LIN {X 0,Y 134.923,Z 410.508,A -85,B 0,C 180,E1 -24681.385,E2 -24681.385} C_VEL
LIN {X 0,Y 135.857,Z 404.738,A -85,B 0,C 180,E1 -24688.426,E2 -24688.426} C_VEL
LIN {X 0,Y 136.109,Z 403.534,A -85,B 0,C 180,E1 -24689.947,E2 -24689.947} C_VEL
LIN {X 0,Y 136.386,Z 403.497,A -85,B 0,C 180,E1 -24691.018,E2 -24691.018} C_VEL
LIN {X 0,Y 136.277,Z 403.499,A -85,B 0,C 180,E1 -24694.562,E2 -24694.562} C_VEL
LIN {X 0,Y 136.081,Z 403.534,A -85,B 0,C 180,E1 -24699.223,E2 -24699.223} C_VEL
LIN {X 0,Y 136.001,Z 403.539,A -85,B 0,C 180,E1 -24703.658,E2 -24703.658} C_VEL
LIN {X 0,Y 136.007,Z 403.542,A -85,B 0,C 180,E1 -24707.797,E2 -24707.797} C_VEL
LIN {X 0,Y 136.029,Z 403.534,A -85,B 0,C 180,E1 -24711.684,E2 -24711.684} C_VEL
LIN {X 0,Y 136.087,Z 403.533,A -85,B 0,C 180,E1 -24715.721,E2 -24715.721} C_VEL
LIN {X 0,Y 136.149,Z 403.524,A -85,B 0,C 180,E1 -24722.317,E2 -24722.317} C_VEL
LIN {X 0,Y 136.247,Z 403.508,A -85,B 0,C 180,E1 -24728.833,E2 -24728.833} C_VEL
LIN {X 0,Y 136.275,Z 403.507,A -85,B 0,C 180,E1 -24735.057,E2 -24735.057} C_VEL
LIN {X 0,Y 136.447,Z 403.483,A -85,B 0,C 180,E1 -24738.138,E2 -24738.138} C_VEL
LIN {X 0,Y 136.555,Z 403.474,A -85,B 0,C 180,E1 -24741.118,E2 -24741.118} C_VEL
LIN {X 0,Y 137.136,Z 403.404,A -85,B 0,C 180,E1 -24750,E2 -24750} C_VEL
LIN {X 0,Y 136.595,Z 403.469,A -85,B 0,C 180,E1 -24758.879,E2 -24758.879} C_VEL
LIN {X 0,Y 136.493,Z 403.477,A -85,B 0,C 180,E1 -24761.954,E2 -24761.954} C_VEL
LIN {X 0,Y 136.276,Z 403.509,A -85,B 0,C 180,E1 -24768.025,E2 -24768.025} C_VEL
LIN {X 0,Y 136.229,Z 403.51,A -85,B 0,C 180,E1 -24771.779,E2 -24771.779} C_VEL
LIN {X 0,Y 136.103,Z 403.528,A -85,B 0,C 180,E1 -24778.616,E2 -24778.616} C_VEL
LIN {X 0,Y 136.081,Z 403.533,A -85,B 0,C 180,E1 -24784.618,E2 -24784.618} C_VEL
LIN {X 0,Y 136.052,Z 403.532,A -85,B 0,C 180,E1 -24789.208,E2 -24789.208} C_VEL
LIN {X 0,Y 135.999,Z 403.544,A -85,B 0,C 180,E1 -24793.657,E2 -24793.657} C_VEL
LIN {X 0,Y 135.985,Z 403.541,A -85,B 0,C 180,E1 -24797.788,E2 -24797.788} C_VEL
LIN {X 0,Y 136.029,Z 403.54,A -85,B 0,C 180,E1 -24801.684,E2 -24801.684} C_VEL
LIN {X 0,Y 136.058,Z 403.53,A -85,B 0,C 180,E1 -24805.738,E2 -24805.738} C_VEL
LIN {X 0,Y 136.149,Z 403.524,A -85,B 0,C 180,E1 -24812.317,E2 -24812.317} C_VEL
LIN {X 0,Y 136.246,Z 403.515,A -85,B 0,C 180,E1 -24818.833,E2 -24818.833} C_VEL
LIN {X 0,Y 136.291,Z 403.507,A -85,B 0,C 180,E1 -24825.058,E2 -24825.058} C_VEL
LIN {X 0,Y 136.503,Z 403.481,A -85,B 0,C 180,E1 -24828.115,E2 -24828.115} C_VEL
LIN {X 0,Y 136.61,Z 403.461,A -85,B 0,C 180,E1 -24831.121,E2 -24831.121} C_VEL
LIN {X 0,Y 137.136,Z 403.396,A -85,B 0,C 180,E1 -24840,E2 -24840} C_VEL
LIN {X 0,Y 136.61,Z 403.463,A -85,B 0,C 180,E1 -24848.878,E2 -24848.878} C_VEL
LIN {X 0,Y 136.494,Z 403.482,A -85,B 0,C 180,E1 -24851.958,E2 -24851.958} C_VEL
LIN {X 0,Y 136.253,Z 403.507,A -85,B 0,C 180,E1 -24858.028,E2 -24858.028} C_VEL
LIN {X 0,Y 136.199,Z 403.52,A -85,B 0,C 180,E1 -24861.749,E2 -24861.749} C_VEL
LIN {X 0,Y 136.101,Z 403.531,A -85,B 0,C 180,E1 -24868.616,E2 -24868.616} C_VEL
LIN {X 0,Y 136.079,Z 403.529,A -85,B 0,C 180,E1 -24874.618,E2 -24874.618} C_VEL
LIN {X 0,Y 136.063,Z 403.536,A -85,B 0,C 180,E1 -24879.214,E2 -24879.214} C_VEL
LIN {X 0,Y 136.313,Z 403.581,A -85,B 0,C 180,E1 -24885.161,E2 -24885.161} C_VEL
LIN {X 0,Y 137.773,Z 409.554,A -85,B 0,C 180,E1 -24891.226,E2 -24891.226} C_VEL
LIN {X 0,Y 139.191,Z 414.655,A -85,B 0,C 180,E1 -24896.261,E2 -24896.261} C_VEL
LIN {X 0,Y 139.438,Z 416.517,A -85,B 0,C 180,E1 -24898.049,E2 -24898.049} C_VEL
LIN {X 0,Y 136.371,Z 425.684,A -85,B 0,C 180,E1 -24907.203,E2 -24907.203} C_VEL
LIN {X 0,Y 136.444,Z 432.258,A -85,B 0,C 180,E1 -24913.927,E2 -24913.927} C_VEL
LIN {X 0,Y 136.598,Z 432.809,A -85,B 0,C 180,E1 -24914.234,E2 -24914.234} C_VEL
LIN {X 0,Y 137.103,Z 444.83,A -85,B 0,C 180,E1 -24915.94,E2 -24915.94} C_VEL
LIN {X 0,Y 138.431,Z 457.423,A -85,B 0,C 180,E1 -24918.283,E2 -24918.283} C_VEL
LIN {X 0,Y 139.405,Z 464.257,A -85,B 0,C 180,E1 -24919.837,E2 -24919.837} C_VEL
LIN {X 0,Y 139.365,Z 473.819,A -85,B 0,C 180,E1 -24922.758,E2 -24922.758} C_VEL
LIN {X 0,Y 139.631,Z 483.352,A -85,B 0,C 180,E1 -24926.393,E2 -24926.393} C_VEL
LIN {X 0,Y 140.17,Z 490.988,A -85,B 0,C 180,E1 -24930,E2 -24930} C_VEL
LIN {X 0,Y 140.133,Z 494.562,A -85,B 0,C 180,E1 -24932.156,E2 -24932.156} C_VEL
LIN {X 0,Y 139.561,Z 497.394,A -85,B 0,C 180,E1 -24934.332,E2 -24934.332} C_VEL
LIN {X 0,Y 138.249,Z 501.754,A -85,B 0,C 180,E1 -24938.773,E2 -24938.773} C_VEL
LIN {X 0,Y 137.884,Z 506.27,A -85,B 0,C 180,E1 -24944.765,E2 -24944.765} C_VEL
LIN {X 0,Y 139.405,Z 509.537,A -85,B 0,C 180,E1 -24950.665,E2 -24950.665} C_VEL
LIN {X 0,Y 142.833,Z 511.707,A -85,B 0,C 180,E1 -24956.286,E2 -24956.286} C_VEL
LIN {X 0,Y 148.061,Z 512.881,A -85,B 0,C 180,E1 -24961.476,E2 -24961.476} C_VEL
LIN {X 0,Y 154.895,Z 513.043,A -85,B 0,C 180,E1 -24966.146,E2 -24966.146} C_VEL
LIN {X 0,Y 163.095,Z 512.189,A -85,B 0,C 180,E1 -24970.269,E2 -24970.269} C_VEL
LIN {X 0,Y 172.559,Z 510.242,A -85,B 0,C 180,E1 -24973.819,E2 -24973.819} C_VEL
LIN {X 0,Y 177.592,Z 508.832,A -85,B 0,C 180,E1 -24975.425,E2 -24975.425} C_VEL
LIN {X 0,Y 179.65,Z 508.061,A -85,B 0,C 180,E1 -24976.364,E2 -24976.364} C_VEL
LIN {X 0,Y 180.102,Z 507.363,A -85,B 0,C 180,E1 -24977.853,E2 -24977.853} C_VEL
LIN {X 0,Y 178.396,Z 506.566,A -85,B 0,C 180,E1 -24980.926,E2 -24980.926} C_VEL
LIN {X 0,Y 176.25,Z 506.125,A -85,B 0,C 180,E1 -24983.264,E2 -24983.264} C_VEL
LIN {X 0,Y 172.11,Z 506.046,A -85,B 0,C 180,E1 -24985.132,E2 -24985.132} C_VEL
LIN {X 0,Y 165.014,Z 505.378,A -85,B 0,C 180,E1 -24987.834,E2 -24987.834} C_VEL
LIN {X 0,Y 158.459,Z 503.885,A -85,B 0,C 180,E1 -24990.799,E2 -24990.799} C_VEL
LIN {X 0,Y 154.466,Z 502.309,A -85,B 0,C 180,E1 -24992.936,E2 -24992.936} C_VEL
LIN {X 0,Y 149.037,Z 499.137,A -85,B 0,C 180,E1 -24996.37,E2 -24996.37} C_VEL
LIN {X 0,Y 148.231,Z 498.488,A -85,B 0,C 180,E1 -24996.975,E2 -24996.975} C_VEL
LIN {X 0,Y 145.275,Z 496.327,A -85,B 0,C 180,E1 -24998.773,E2 -24998.773} C_VEL
LIN {X 0,Y 139.381,Z 491.98,A -85,B 0,C 180,E1 -25001.462,E2 -25001.462} C_VEL
LIN {X 0,Y 134.104,Z 486.835,A -85,B 0,C 180,E1 -25004.254,E2 -25004.254} C_VEL
LIN {X 0,Y 132.202,Z 483.453,A -85,B 0,C 180,E1 -25006.182,E2 -25006.182} C_VEL
LIN {X 0,Y 130.071,Z 474.061,A -85,B 0,C 180,E1 -25011.455,E2 -25011.455} C_VEL
LIN {X 0,Y 129.418,Z 465.891,A -85,B 0,C 180,E1 -25015.328,E2 -25015.328} C_VEL
LIN {X 0,Y 129.469,Z 454.926,A -85,B 0,C 180,E1 -25019.611,E2 -25019.611} C_VEL
LIN {X 0,Y 129.665,Z 446.445,A -85,B 0,C 180,E1 -25022.33,E2 -25022.33} C_VEL
LIN {X 0,Y 129.871,Z 436.015,A -85,B 0,C 180,E1 -25025.045,E2 -25025.045} C_VEL
LIN {X 0,Y 129.845,Z 430.527,A -85,B 0,C 180,E1 -25026.215,E2 -25026.215} C_VEL
LIN {X 0,Y 128.67,Z 421.434,A -85,B 0,C 180,E1 -25027.782,E2 -25027.782} C_VEL
LIN {X 0,Y 127.321,Z 417.429,A -85,B 0,C 180,E1 -25032.756,E2 -25032.756} C_VEL
LIN {X 0,Y 127.758,Z 411.164,A -85,B 0,C 180,E1 -25040.743,E2 -25040.743} C_VEL
LIN {X 0,Y 128.612,Z 405.807,A -85,B 0,C 180,E1 -25047.602,E2 -25047.602} C_VEL
LIN {X 0,Y 128.89,Z 404.435,A -85,B 0,C 180,E1 -25049.39,E2 -25049.39} C_VEL
LIN {X 0,Y 129.242,Z 404.372,A -85,B 0,C 180,E1 -25052.942,E2 -25052.942} C_VEL
LIN {X 0,Y 129.073,Z 404.406,A -85,B 0,C 180,E1 -25056.795,E2 -25056.795} C_VEL
LIN {X 0,Y 128.985,Z 404.415,A -85,B 0,C 180,E1 -25060.833,E2 -25060.833} C_VEL
LIN {X 0,Y 128.924,Z 404.425,A -85,B 0,C 180,E1 -25065.127,E2 -25065.127} C_VEL
LIN {X 0,Y 128.944,Z 404.42,A -85,B 0,C 180,E1 -25069.735,E2 -25069.735} C_VEL
LIN {X 0,Y 128.983,Z 404.419,A -85,B 0,C 180,E1 -25074.818,E2 -25074.818} C_VEL
LIN {X 0,Y 129.036,Z 404.406,A -85,B 0,C 180,E1 -25080.647,E2 -25080.647} C_VEL
LIN {X 0,Y 129.111,Z 404.398,A -85,B 0,C 180,E1 -25087.602,E2 -25087.602} C_VEL
LIN {X 0,Y 129.16,Z 404.395,A -85,B 0,C 180,E1 -25090.944,E2 -25090.944} C_VEL
LIN {X 0,Y 129.369,Z 404.364,A -85,B 0,C 180,E1 -25097.922,E2 -25097.922} C_VEL
LIN {X 0,Y 129.48,Z 404.356,A -85,B 0,C 180,E1 -25100.628,E2 -25100.628} C_VEL
LIN {X 0,Y 130.091,Z 404.281,A -85,B 0,C 180,E1 -25110,E2 -25110} C_VEL
LIN {X 0,Y 129.52,Z 404.351,A -85,B 0,C 180,E1 -25119.368,E2 -25119.368} C_VEL
LIN {X 0,Y 129.397,Z 404.359,A -85,B 0,C 180,E1 -25122.548,E2 -25122.548} C_VEL
LIN {X 0,Y 129.188,Z 404.391,A -85,B 0,C 180,E1 -25129.051,E2 -25129.051} C_VEL
LIN {X 0,Y 129.138,Z 404.395,A -85,B 0,C 180,E1 -25132.393,E2 -25132.393} C_VEL
LIN {X 0,Y 129.037,Z 404.406,A -85,B 0,C 180,E1 -25139.373,E2 -25139.373} C_VEL
LIN {X 0,Y 128.994,Z 404.418,A -85,B 0,C 180,E1 -25145.189,E2 -25145.189} C_VEL
LIN {X 0,Y 128.952,Z 404.42,A -85,B 0,C 180,E1 -25150.845,E2 -25150.845} C_VEL
LIN {X 0,Y 128.917,Z 404.424,A -85,B 0,C 180,E1 -25155.129,E2 -25155.129} C_VEL
LIN {X 0,Y 128.937,Z 404.423,A -85,B 0,C 180,E1 -25159.738,E2 -25159.738} C_VEL
LIN {X 0,Y 128.962,Z 404.416,A -85,B 0,C 180,E1 -25164.83,E2 -25164.83} C_VEL
LIN {X 0,Y 129.052,Z 404.41,A -85,B 0,C 180,E1 -25170.651,E2 -25170.651} C_VEL
LIN {X 0,Y 129.109,Z 404.402,A -85,B 0,C 180,E1 -25177.727,E2 -25177.727} C_VEL
LIN {X 0,Y 129.165,Z 404.393,A -85,B 0,C 180,E1 -25180.945,E2 -25180.945} C_VEL
LIN {X 0,Y 129.42,Z 404.363,A -85,B 0,C 180,E1 -25187.814,E2 -25187.814} C_VEL
LIN {X 0,Y 129.532,Z 404.344,A -85,B 0,C 180,E1 -25190.632,E2 -25190.632} C_VEL
LIN {X 0,Y 130.092,Z 404.274,A -85,B 0,C 180,E1 -25200,E2 -25200} C_VEL
LIN {X 0,Y 129.532,Z 404.344,A -85,B 0,C 180,E1 -25209.368,E2 -25209.368} C_VEL
LIN {X 0,Y 129.395,Z 404.367,A -85,B 0,C 180,E1 -25212.548,E2 -25212.548} C_VEL
LIN {X 0,Y 129.161,Z 404.393,A -85,B 0,C 180,E1 -25219.055,E2 -25219.055} C_VEL
LIN {X 0,Y 129.109,Z 404.402,A -85,B 0,C 180,E1 -25222.398,E2 -25222.398} C_VEL
LIN {X 0,Y 129.036,Z 404.411,A -85,B 0,C 180,E1 -25229.373,E2 -25229.373} C_VEL
LIN {X 0,Y 128.994,Z 404.411,A -85,B 0,C 180,E1 -25235.19,E2 -25235.19} C_VEL
LIN {X 0,Y 129.011,Z 404.412,A -85,B 0,C 180,E1 -25240.822,E2 -25240.822} C_VEL
LIN {X 0,Y 129.309,Z 404.45,A -85,B 0,C 180,E1 -25245.452,E2 -25245.452} C_VEL
LIN {X 0,Y 130.772,Z 410.28,A -85,B 0,C 180,E1 -25251.707,E2 -25251.707} C_VEL
LIN {X 0,Y 131.968,Z 414.402,A -85,B 0,C 180,E1 -25256.001,E2 -25256.001} C_VEL
LIN {X 0,Y 132.301,Z 416.274,A -85,B 0,C 180,E1 -25257.913,E2 -25257.913} C_VEL
LIN {X 0,Y 129.245,Z 425.368,A -85,B 0,C 180,E1 -25267.627,E2 -25267.627} C_VEL
LIN {X 0,Y 129.433,Z 431.429,A -85,B 0,C 180,E1 -25274.247,E2 -25274.247} C_VEL
LIN {X 0,Y 129.83,Z 432.468,A -85,B 0,C 180,E1 -25275.124,E2 -25275.124} C_VEL
LIN {X 0,Y 130.443,Z 444.677,A -85,B 0,C 180,E1 -25276.986,E2 -25276.986} C_VEL
LIN {X 0,Y 131.772,Z 456.247,A -85,B 0,C 180,E1 -25279.242,E2 -25279.242} C_VEL
LIN {X 0,Y 132.84,Z 463.183,A -85,B 0,C 180,E1 -25280.868,E2 -25280.868} C_VEL
LIN {X 0,Y 132.91,Z 473.806,A -85,B 0,C 180,E1 -25284.31,E2 -25284.31} C_VEL
LIN {X 0,Y 133.271,Z 482.289,A -85,B 0,C 180,E1 -25287.734,E2 -25287.734} C_VEL
LIN {X 0,Y 133.772,Z 488.453,A -85,B 0,C 180,E1 -25290.753,E2 -25290.753} C_VEL
LIN {X 0,Y 133.736,Z 492.301,A -85,B 0,C 180,E1 -25293.165,E2 -25293.165} C_VEL
LIN {X 0,Y 132.794,Z 495.697,A -85,B 0,C 180,E1 -25296.076,E2 -25296.076} C_VEL
LIN {X 0,Y 131.466,Z 501.251,A -85,B 0,C 180,E1 -25302.347,E2 -25302.347} C_VEL
LIN {X 0,Y 132.063,Z 505.446,A -85,B 0,C 180,E1 -25308.621,E2 -25308.621} C_VEL
LIN {X 0,Y 134.734,Z 508.516,A -85,B 0,C 180,E1 -25314.664,E2 -25314.664} C_VEL
LIN {X 0,Y 139.237,Z 510.545,A -85,B 0,C 180,E1 -25320.315,E2 -25320.315} C_VEL
LIN {X 0,Y 145.557,Z 511.616,A -85,B 0,C 180,E1 -25325.409,E2 -25325.409} C_VEL
LIN {X 0,Y 153.433,Z 511.739,A -85,B 0,C 180,E1 -25329.887,E2 -25329.887} C_VEL
LIN {X 0,Y 162.537,Z 510.85,A -85,B 0,C 180,E1 -25333.776,E2 -25333.776} C_VEL
LIN {X 0,Y 172.611,Z 508.879,A -85,B 0,C 180,E1 -25337.129,E2 -25337.129} C_VEL
LIN {X 0,Y 172.25,Z 508.109,A -85,B 0,C 180,E1 -25339.246,E2 -25339.246} C_VEL
LIN {X 0,Y 170.406,Z 507.374,A -85,B 0,C 180,E1 -25341.783,E2 -25341.783} C_VEL
LIN {X 0,Y 166.321,Z 506.966,A -85,B 0,C 180,E1 -25343.731,E2 -25343.731} C_VEL
LIN {X 0,Y 156.711,Z 505.324,A -85,B 0,C 180,E1 -25347.441,E2 -25347.441} C_VEL
LIN {X 0,Y 152.284,Z 503.896,A -85,B 0,C 180,E1 -25349.492,E2 -25349.492} C_VEL
LIN {X 0,Y 144.308,Z 499.738,A -85,B 0,C 180,E1 -25354.004,E2 -25354.004} C_VEL
LIN {X 0,Y 139.337,Z 495.438,A -85,B 0,C 180,E1 -25357.772,E2 -25357.772} C_VEL
LIN {X 0,Y 134.671,Z 489.065,A -85,B 0,C 180,E1 -25362.538,E2 -25362.538} C_VEL
LIN {X 0,Y 132.202,Z 483.453,A -85,B 0,C 180,E1 -25366.182,E2 -25366.182} C_VEL
LIN {X 0,Y 130.599,Z 479.926,A -85,B 0,C 180,E1 -25368.095,E2 -25368.095} C_VEL
LIN {X 0,Y 126.875,Z 473.349,A -85,B 0,C 180,E1 -25370.916,E2 -25370.916} C_VEL
LIN {X 0,Y 123.597,Z 466.089,A -85,B 0,C 180,E1 -25373.694,E2 -25373.694} C_VEL
LIN {X 0,Y 122.777,Z 461.607,A -85,B 0,C 180,E1 -25375.504,E2 -25375.504} C_VEL
LIN {X 0,Y 122.912,Z 450.852,A -85,B 0,C 180,E1 -25379.591,E2 -25379.591} C_VEL
LIN {X 0,Y 122.991,Z 441.44,A -85,B 0,C 180,E1 -25382.457,E2 -25382.457} C_VEL
LIN {X 0,Y 123.165,Z 430.67,A -85,B 0,C 180,E1 -25385.116,E2 -25385.116} C_VEL
LIN {X 0,Y 121.993,Z 421.815,A -85,B 0,C 180,E1 -25386.696,E2 -25386.696} C_VEL
LIN {X 0,Y 120.327,Z 417.894,A -85,B 0,C 180,E1 -25391.796,E2 -25391.796} C_VEL
LIN {X 0,Y 120.699,Z 410.831,A -85,B 0,C 180,E1 -25401.307,E2 -25401.307} C_VEL
LIN {X 0,Y 121.656,Z 405.488,A -85,B 0,C 180,E1 -25408.513,E2 -25408.513} C_VEL
LIN {X 0,Y 121.964,Z 405.294,A -85,B 0,C 180,E1 -25411.24,E2 -25411.24} C_VEL
LIN {X 0,Y 122.046,Z 405.279,A -85,B 0,C 180,E1 -25416.274,E2 -25416.274} C_VEL
LIN {X 0,Y 121.91,Z 405.295,A -85,B 0,C 180,E1 -25421.457,E2 -25421.457} C_VEL
LIN {X 0,Y 121.874,Z 405.303,A -85,B 0,C 180,E1 -25428.561,E2 -25428.561} C_VEL
LIN {X 0,Y 121.935,Z 405.297,A -85,B 0,C 180,E1 -25434.804,E2 -25434.804} C_VEL
LIN {X 0,Y 121.943,Z 405.288,A -85,B 0,C 180,E1 -25439.827,E2 -25439.827} C_VEL
LIN {X 0,Y 121.986,Z 405.288,A -85,B 0,C 180,E1 -25446.215,E2 -25446.215} C_VEL
LIN {X 0,Y 122.05,Z 405.277,A -85,B 0,C 180,E1 -25449.787,E2 -25449.787} C_VEL
LIN {X 0,Y 122.242,Z 405.25,A -85,B 0,C 180,E1 -25456.704,E2 -25456.704} C_VEL
LIN {X 0,Y 122.409,Z 405.236,A -85,B 0,C 180,E1 -25460.081,E2 -25460.081} C_VEL
LIN {X 0,Y 122.602,Z 405.209,A -85,B 0,C 180,E1 -25466.714,E2 -25466.714} C_VEL
LIN {X 0,Y 123.045,Z 405.159,A -85,B 0,C 180,E1 -25470,E2 -25470} C_VEL
LIN {X 0,Y 122.45,Z 405.231,A -85,B 0,C 180,E1 -25476.591,E2 -25476.591} C_VEL
LIN {X 0,Y 122.449,Z 405.231,A -85,B 0,C 180,E1 -25479.915,E2 -25479.915} C_VEL
LIN {X 0,Y 122.289,Z 405.245,A -85,B 0,C 180,E1 -25483.29,E2 -25483.29} C_VEL
LIN {X 0,Y 122.076,Z 405.273,A -85,B 0,C 180,E1 -25490.208,E2 -25490.208} C_VEL
LIN {X 0,Y 121.998,Z 405.287,A -85,B 0,C 180,E1 -25493.781,E2 -25493.781} C_VEL
LIN {X 0,Y 121.943,Z 405.288,A -85,B 0,C 180,E1 -25500.173,E2 -25500.173} C_VEL
LIN {X 0,Y 121.913,Z 405.297,A -85,B 0,C 180,E1 -25506.189,E2 -25506.189} C_VEL
LIN {X 0,Y 121.885,Z 405.302,A -85,B 0,C 180,E1 -25511.444,E2 -25511.444} C_VEL
LIN {X 0,Y 121.866,Z 405.3,A -85,B 0,C 180,E1 -25518.565,E2 -25518.565} C_VEL
LIN {X 0,Y 121.914,Z 405.294,A -85,B 0,C 180,E1 -25524.797,E2 -25524.797} C_VEL
LIN {X 0,Y 121.94,Z 405.295,A -85,B 0,C 180,E1 -25529.828,E2 -25529.828} C_VEL
LIN {X 0,Y 121.985,Z 405.287,A -85,B 0,C 180,E1 -25536.215,E2 -25536.215} C_VEL
LIN {X 0,Y 122.053,Z 405.28,A -85,B 0,C 180,E1 -25539.788,E2 -25539.788} C_VEL
LIN {X 0,Y 122.288,Z 405.253,A -85,B 0,C 180,E1 -25546.709,E2 -25546.709} C_VEL
LIN {X 0,Y 122.458,Z 405.228,A -85,B 0,C 180,E1 -25550.086,E2 -25550.086} C_VEL
LIN {X 0,Y 122.612,Z 405.211,A -85,B 0,C 180,E1 -25556.714,E2 -25556.714} C_VEL
LIN {X 0,Y 123.046,Z 405.151,A -85,B 0,C 180,E1 -25560,E2 -25560} C_VEL
LIN {X 0,Y 122.459,Z 405.228,A -85,B 0,C 180,E1 -25566.591,E2 -25566.591} C_VEL
LIN {X 0,Y 122.458,Z 405.226,A -85,B 0,C 180,E1 -25569.914,E2 -25569.914} C_VEL
LIN {X 0,Y 122.265,Z 405.254,A -85,B 0,C 180,E1 -25573.293,E2 -25573.293} C_VEL
LIN {X 0,Y 122.051,Z 405.282,A -85,B 0,C 180,E1 -25580.212,E2 -25580.212} C_VEL
LIN {X 0,Y 121.984,Z 405.288,A -85,B 0,C 180,E1 -25583.784,E2 -25583.784} C_VEL
LIN {X 0,Y 121.942,Z 405.296,A -85,B 0,C 180,E1 -25590.174,E2 -25590.174} C_VEL
LIN {X 0,Y 121.916,Z 405.296,A -85,B 0,C 180,E1 -25596.192,E2 -25596.192} C_VEL
LIN {X 0,Y 122.073,Z 405.273,A -85,B 0,C 180,E1 -25603.698,E2 -25603.698} C_VEL
LIN {X 0,Y 122.297,Z 405.278,A -85,B 0,C 180,E1 -25605.79,E2 -25605.79} C_VEL
LIN {X 0,Y 123.862,Z 411.27,A -85,B 0,C 180,E1 -25612.596,E2 -25612.596} C_VEL
LIN {X 0,Y 125.082,Z 415.684,A -85,B 0,C 180,E1 -25617.438,E2 -25617.438} C_VEL
LIN {X 0,Y 123.854,Z 419.021,A -85,B 0,C 180,E1 -25621.163,E2 -25621.163} C_VEL
LIN {X 0,Y 122.14,Z 429.42,A -85,B 0,C 180,E1 -25633.28,E2 -25633.28} C_VEL
LIN {X 0,Y 123.086,Z 431.907,A -85,B 0,C 180,E1 -25636.089,E2 -25636.089} C_VEL
LIN {X 0,Y 123.909,Z 445.534,A -85,B 0,C 180,E1 -25638.343,E2 -25638.343} C_VEL
LIN {X 0,Y 125.437,Z 456.947,A -85,B 0,C 180,E1 -25640.731,E2 -25640.731} C_VEL
LIN {X 0,Y 126.306,Z 462.085,A -85,B 0,C 180,E1 -25642.004,E2 -25642.004} C_VEL
LIN {X 0,Y 126.499,Z 472.65,A -85,B 0,C 180,E1 -25645.619,E2 -25645.619} C_VEL
LIN {X 0,Y 127.048,Z 481.337,A -85,B 0,C 180,E1 -25649.368,E2 -25649.368} C_VEL
LIN {X 0,Y 127.589,Z 487.079,A -85,B 0,C 180,E1 -25652.368,E2 -25652.368} C_VEL
LIN {X 0,Y 127.359,Z 489.743,A -85,B 0,C 180,E1 -25654.193,E2 -25654.193} C_VEL
LIN {X 0,Y 126.124,Z 493.904,A -85,B 0,C 180,E1 -25658.008,E2 -25658.008} C_VEL
LIN {X 0,Y 125.217,Z 499.381,A -85,B 0,C 180,E1 -25664.63,E2 -25664.63} C_VEL
LIN {X 0,Y 125.873,Z 502.645,A -85,B 0,C 180,E1 -25669.573,E2 -25669.573} C_VEL
LIN {X 0,Y 128.681,Z 506.08,A -85,B 0,C 180,E1 -25675.908,E2 -25675.908} C_VEL
LIN {X 0,Y 133.412,Z 508.447,A -85,B 0,C 180,E1 -25681.789,E2 -25681.789} C_VEL
LIN {X 0,Y 139.98,Z 509.929,A -85,B 0,C 180,E1 -25687.048,E2 -25687.048} C_VEL
LIN {X 0,Y 148.135,Z 510.49,A -85,B 0,C 180,E1 -25691.622,E2 -25691.622} C_VEL
LIN {X 0,Y 157.516,Z 510.086,A -85,B 0,C 180,E1 -25695.552,E2 -25695.552} C_VEL
LIN {X 0,Y 165.089,Z 509.134,A -85,B 0,C 180,E1 -25698.046,E2 -25698.046} C_VEL
LIN {X 0,Y 164.109,Z 508.288,A -85,B 0,C 180,E1 -25700.431,E2 -25700.431} C_VEL
LIN {X 0,Y 160.623,Z 507.645,A -85,B 0,C 180,E1 -25702.225,E2 -25702.225} C_VEL
LIN {X 0,Y 150.747,Z 505.383,A -85,B 0,C 180,E1 -25705.982,E2 -25705.982} C_VEL
LIN {X 0,Y 144.014,Z 502.65,A -85,B 0,C 180,E1 -25709.176,E2 -25709.176} C_VEL
LIN {X 0,Y 137.971,Z 498.908,A -85,B 0,C 180,E1 -25712.713,E2 -25712.713} C_VEL
LIN {X 0,Y 132.851,Z 494.204,A -85,B 0,C 180,E1 -25716.624,E2 -25716.624} C_VEL
LIN {X 0,Y 128.073,Z 487.269,A -85,B 0,C 180,E1 -25721.607,E2 -25721.607} C_VEL
LIN {X 0,Y 125.145,Z 480.069,A -85,B 0,C 180,E1 -25726.192,E2 -25726.192} C_VEL
LIN {X 0,Y 123.428,Z 471.271,A -85,B 0,C 180,E1 -25730.992,E2 -25730.992} C_VEL
LIN {X 0,Y 122.777,Z 461.607,A -85,B 0,C 180,E1 -25735.504,E2 -25735.504} C_VEL
LIN {X 0,Y 122.092,Z 457.024,A -85,B 0,C 180,E1 -25737.205,E2 -25737.205} C_VEL
LIN {X 0,Y 120.672,Z 452.145,A -85,B 0,C 180,E1 -25738.65,E2 -25738.65} C_VEL
LIN {X 0,Y 117.434,Z 441.865,A -85,B 0,C 180,E1 -25741.172,E2 -25741.172} C_VEL
LIN {X 0,Y 116.552,Z 436.486,A -85,B 0,C 180,E1 -25742.448,E2 -25742.448} C_VEL
LIN {X 0,Y 116.494,Z 434.675,A -85,B 0,C 180,E1 -25742.895,E2 -25742.895} C_VEL
LIN {X 0,Y 116.409,Z 429.421,A -85,B 0,C 180,E1 -25744.112,E2 -25744.112} C_VEL
LIN {X 0,Y 115.383,Z 422.175,A -85,B 0,C 180,E1 -25745.462,E2 -25745.462} C_VEL
LIN {X 0,Y 113.392,Z 418.319,A -85,B 0,C 180,E1 -25750.716,E2 -25750.716} C_VEL
LIN {X 0,Y 113.674,Z 410.429,A -85,B 0,C 180,E1 -25761.968,E2 -25761.968} C_VEL
LIN {X 0,Y 114.475,Z 406.23,A -85,B 0,C 180,E1 -25768.162,E2 -25768.162} C_VEL
LIN {X 0,Y 114.898,Z 406.174,A -85,B 0,C 180,E1 -25771.09,E2 -25771.09} C_VEL
LIN {X 0,Y 114.922,Z 406.17,A -85,B 0,C 180,E1 -25777.343,E2 -25777.343} C_VEL
LIN {X 0,Y 114.811,Z 406.177,A -85,B 0,C 180,E1 -25782.729,E2 -25782.729} C_VEL
LIN {X 0,Y 114.797,Z 406.185,A -85,B 0,C 180,E1 -25787.667,E2 -25787.667} C_VEL
LIN {X 0,Y 114.8,Z 406.18,A -85,B 0,C 180,E1 -25792.737,E2 -25792.737} C_VEL
LIN {X 0,Y 114.869,Z 406.17,A -85,B 0,C 180,E1 -25798.933,E2 -25798.933} C_VEL
LIN {X 0,Y 114.949,Z 406.163,A -85,B 0,C 180,E1 -25806.507,E2 -25806.507} C_VEL
LIN {X 0,Y 115.016,Z 406.158,A -85,B 0,C 180,E1 -25812.21,E2 -25812.21} C_VEL
LIN {X 0,Y 115.254,Z 406.12,A -85,B 0,C 180,E1 -25817.333,E2 -25817.333} C_VEL
LIN {X 0,Y 115.369,Z 406.112,A -85,B 0,C 180,E1 -25823.002,E2 -25823.002} C_VEL
LIN {X 0,Y 115.996,Z 406.037,A -85,B 0,C 180,E1 -25830,E2 -25830} C_VEL
LIN {X 0,Y 115.391,Z 406.11,A -85,B 0,C 180,E1 -25836.996,E2 -25836.996} C_VEL
LIN {X 0,Y 115.308,Z 406.114,A -85,B 0,C 180,E1 -25842.785,E2 -25842.785} C_VEL
LIN {X 0,Y 115.036,Z 406.156,A -85,B 0,C 180,E1 -25847.786,E2 -25847.786} C_VEL
LIN {X 0,Y 114.968,Z 406.161,A -85,B 0,C 180,E1 -25853.514,E2 -25853.514} C_VEL
LIN {X 0,Y 114.87,Z 406.17,A -85,B 0,C 180,E1 -25861.068,E2 -25861.068} C_VEL
LIN {X 0,Y 114.803,Z 406.178,A -85,B 0,C 180,E1 -25867.747,E2 -25867.747} C_VEL
LIN {X 0,Y 114.794,Z 406.185,A -85,B 0,C 180,E1 -25872.72,E2 -25872.72} C_VEL
LIN {X 0,Y 114.789,Z 406.18,A -85,B 0,C 180,E1 -25877.663,E2 -25877.663} C_VEL
LIN {X 0,Y 114.789,Z 406.186,A -85,B 0,C 180,E1 -25882.743,E2 -25882.743} C_VEL
LIN {X 0,Y 114.863,Z 406.177,A -85,B 0,C 180,E1 -25888.937,E2 -25888.937} C_VEL
LIN {X 0,Y 114.948,Z 406.164,A -85,B 0,C 180,E1 -25896.507,E2 -25896.507} C_VEL
LIN {X 0,Y 115.022,Z 406.151,A -85,B 0,C 180,E1 -25902.211,E2 -25902.211} C_VEL
LIN {X 0,Y 115.288,Z 406.124,A -85,B 0,C 180,E1 -25907.257,E2 -25907.257} C_VEL
LIN {X 0,Y 115.395,Z 406.108,A -85,B 0,C 180,E1 -25909.472,E2 -25909.472} C_VEL
LIN {X 0,Y 115.539,Z 406.093,A -85,B 0,C 180,E1 -25916.512,E2 -25916.512} C_VEL
LIN {X 0,Y 115.998,Z 406.029,A -85,B 0,C 180,E1 -25920,E2 -25920} C_VEL
LIN {X 0,Y 115.4,Z 406.106,A -85,B 0,C 180,E1 -25926.996,E2 -25926.996} C_VEL
LIN {X 0,Y 115.394,Z 406.108,A -85,B 0,C 180,E1 -25930.528,E2 -25930.528} C_VEL
LIN {X 0,Y 115.149,Z 406.141,A -85,B 0,C 180,E1 -25934.131,E2 -25934.131} C_VEL
LIN {X 0,Y 114.982,Z 406.162,A -85,B 0,C 180,E1 -25941.514,E2 -25941.514} C_VEL
LIN {X 0,Y 114.871,Z 406.169,A -85,B 0,C 180,E1 -25945.358,E2 -25945.358} C_VEL
LIN {X 0,Y 114.869,Z 406.175,A -85,B 0,C 180,E1 -25951.068,E2 -25951.068} C_VEL
LIN {X 0,Y 114.821,Z 406.182,A -85,B 0,C 180,E1 -25957.74,E2 -25957.74} C_VEL
LIN {X 0,Y 115.331,Z 406.232,A -85,B 0,C 180,E1 -25966.391,E2 -25966.391} C_VEL
LIN {X 0,Y 116.827,Z 411.721,A -85,B 0,C 180,E1 -25973.017,E2 -25973.017} C_VEL
LIN {X 0,Y 117.906,Z 415.607,A -85,B 0,C 180,E1 -25977.557,E2 -25977.557} C_VEL
LIN {X 0,Y 115.681,Z 421.588,A -85,B 0,C 180,E1 -25984.832,E2 -25984.832} C_VEL
LIN {X 0,Y 115.225,Z 428.905,A -85,B 0,C 180,E1 -25994.07,E2 -25994.07} C_VEL
LIN {X 0,Y 116.432,Z 431.559,A -85,B 0,C 180,E1 -25997.25,E2 -25997.25} C_VEL
LIN {X 0,Y 117.389,Z 445.011,A -85,B 0,C 180,E1 -25999.653,E2 -25999.653} C_VEL
LIN {X 0,Y 119.201,Z 457.192,A -85,B 0,C 180,E1 -26002.377,E2 -26002.377} C_VEL
LIN {X 0,Y 119.939,Z 461.873,A -85,B 0,C 180,E1 -26003.65,E2 -26003.65} C_VEL
LIN {X 0,Y 120.245,Z 471.274,A -85,B 0,C 180,E1 -26007.082,E2 -26007.082} C_VEL
LIN {X 0,Y 120.895,Z 479.648,A -85,B 0,C 180,E1 -26010.833,E2 -26010.833} C_VEL
LIN {X 0,Y 121.397,Z 484.307,A -85,B 0,C 180,E1 -26013.319,E2 -26013.319} C_VEL
LIN {X 0,Y 121.009,Z 487.259,A -85,B 0,C 180,E1 -26015.498,E2 -26015.498} C_VEL
LIN {X 0,Y 119.315,Z 493.376,A -85,B 0,C 180,E1 -26021.898,E2 -26021.898} C_VEL
LIN {X 0,Y 119.225,Z 497.369,A -85,B 0,C 180,E1 -26027.142,E2 -26027.142} C_VEL
LIN {X 0,Y 121.029,Z 501.66,A -85,B 0,C 180,E1 -26033.984,E2 -26033.984} C_VEL
LIN {X 0,Y 125.006,Z 504.873,A -85,B 0,C 180,E1 -26040.398,E2 -26040.398} C_VEL
LIN {X 0,Y 132.138,Z 507.482,A -85,B 0,C 180,E1 -26047.079,E2 -26047.079} C_VEL
LIN {X 0,Y 138.624,Z 508.616,A -85,B 0,C 180,E1 -26051.23,E2 -26051.23} C_VEL
LIN {X 0,Y 147.696,Z 509.14,A -85,B 0,C 180,E1 -26055.543,E2 -26055.543} C_VEL
LIN {X 0,Y 152.682,Z 509.066,A -85,B 0,C 180,E1 -26057.433,E2 -26057.433} C_VEL
LIN {X 0,Y 157.43,Z 508.649,A -85,B 0,C 180,E1 -26059.369,E2 -26059.369} C_VEL
LIN {X 0,Y 155.029,Z 508.059,A -85,B 0,C 180,E1 -26060.605,E2 -26060.605} C_VEL
LIN {X 0,Y 144.881,Z 505.202,A -85,B 0,C 180,E1 -26064.401,E2 -26064.401} C_VEL
LIN {X 0,Y 135.793,Z 500.718,A -85,B 0,C 180,E1 -26068.832,E2 -26068.832} C_VEL
LIN {X 0,Y 129.908,Z 496.243,A -85,B 0,C 180,E1 -26072.623,E2 -26072.623} C_VEL
LIN {X 0,Y 124.201,Z 489.699,A -85,B 0,C 180,E1 -26077.545,E2 -26077.545} C_VEL
LIN {X 0,Y 120.406,Z 482.784,A -85,B 0,C 180,E1 -26082.155,E2 -26082.155} C_VEL
LIN {X 0,Y 117.573,Z 473.095,A -85,B 0,C 180,E1 -26087.924,E2 -26087.924} C_VEL
LIN {X 0,Y 116.469,Z 462.816,A -85,B 0,C 180,E1 -26093.069,E2 -26093.069} C_VEL
LIN {X 0,Y 116.318,Z 451.278,A -85,B 0,C 180,E1 -26097.836,E2 -26097.836} C_VEL
LIN {X 0,Y 116.374,Z 442.11,A -85,B 0,C 180,E1 -26100.865,E2 -26100.865} C_VEL
LIN {X 0,Y 116.494,Z 434.675,A -85,B 0,C 180,E1 -26102.895,E2 -26102.895} C_VEL
LIN {X 0,Y 115.682,Z 431.022,A -85,B 0,C 180,E1 -26103.73,E2 -26103.73} C_VEL
LIN {X 0,Y 112.941,Z 426.556,A -85,B 0,C 180,E1 -26104.722,E2 -26104.722} C_VEL
LIN {X 0,Y 109.643,Z 422.778,A -85,B 0,C 180,E1 -26105.974,E2 -26105.974} C_VEL
LIN {X 0,Y 107.42,Z 420.303,A -85,B 0,C 180,E1 -26107.506,E2 -26107.506} C_VEL
LIN {X 0,Y 106.756,Z 419.321,A -85,B 0,C 180,E1 -26108.59,E2 -26108.59} C_VEL
LIN {X 0,Y 106.452,Z 411.122,A -85,B 0,C 180,E1 -26120.996,E2 -26120.996} C_VEL
LIN {X 0,Y 107.235,Z 407.129,A -85,B 0,C 180,E1 -26127.308,E2 -26127.308} C_VEL
LIN {X 0,Y 107.848,Z 407.042,A -85,B 0,C 180,E1 -26132.096,E2 -26132.096} C_VEL
LIN {X 0,Y 107.788,Z 407.059,A -85,B 0,C 180,E1 -26138.516,E2 -26138.516} C_VEL
LIN {X 0,Y 107.685,Z 407.07,A -85,B 0,C 180,E1 -26145.883,E2 -26145.883} C_VEL
LIN {X 0,Y 107.696,Z 407.062,A -85,B 0,C 180,E1 -26151.545,E2 -26151.545} C_VEL
LIN {X 0,Y 107.807,Z 407.051,A -85,B 0,C 180,E1 -26158.565,E2 -26158.565} C_VEL
LIN {X 0,Y 107.913,Z 407.038,A -85,B 0,C 180,E1 -26166.998,E2 -26166.998} C_VEL
LIN {X 0,Y 108.034,Z 407.025,A -85,B 0,C 180,E1 -26174.917,E2 -26174.917} C_VEL
LIN {X 0,Y 108.256,Z 406.997,A -85,B 0,C 180,E1 -26178.769,E2 -26178.769} C_VEL
LIN {X 0,Y 108.449,Z 406.97,A -85,B 0,C 180,E1 -26186.284,E2 -26186.284} C_VEL
LIN {X 0,Y 108.946,Z 406.915,A -85,B 0,C 180,E1 -26190,E2 -26190} C_VEL
LIN {X 0,Y 108.331,Z 406.99,A -85,B 0,C 180,E1 -26197.455,E2 -26197.455} C_VEL
LIN {X 0,Y 108.217,Z 406.997,A -85,B 0,C 180,E1 -26203.052,E2 -26203.052} C_VEL
LIN {X 0,Y 107.931,Z 407.039,A -85,B 0,C 180,E1 -26209,E2 -26209} C_VEL
LIN {X 0,Y 107.874,Z 407.047,A -85,B 0,C 180,E1 -26214.201,E2 -26214.201} C_VEL
LIN {X 0,Y 107.796,Z 407.056,A -85,B 0,C 180,E1 -26222.051,E2 -26222.051} C_VEL
LIN {X 0,Y 107.708,Z 407.06,A -85,B 0,C 180,E1 -26228.462,E2 -26228.462} C_VEL
LIN {X 0,Y 107.675,Z 407.067,A -85,B 0,C 180,E1 -26235.887,E2 -26235.887} C_VEL
LIN {X 0,Y 107.688,Z 407.071,A -85,B 0,C 180,E1 -26241.55,E2 -26241.55} C_VEL
LIN {X 0,Y 107.799,Z 407.056,A -85,B 0,C 180,E1 -26248.562,E2 -26248.562} C_VEL
LIN {X 0,Y 107.913,Z 407.042,A -85,B 0,C 180,E1 -26256.998,E2 -26256.998} C_VEL
LIN {X 0,Y 108.048,Z 407.023,A -85,B 0,C 180,E1 -26264.919,E2 -26264.919} C_VEL
LIN {X 0,Y 108.308,Z 406.992,A -85,B 0,C 180,E1 -26268.774,E2 -26268.774} C_VEL
LIN {X 0,Y 108.465,Z 406.975,A -85,B 0,C 180,E1 -26276.285,E2 -26276.285} C_VEL
LIN {X 0,Y 108.948,Z 406.907,A -85,B 0,C 180,E1 -26280,E2 -26280} C_VEL
LIN {X 0,Y 108.342,Z 406.985,A -85,B 0,C 180,E1 -26287.454,E2 -26287.454} C_VEL
LIN {X 0,Y 108.204,Z 407.006,A -85,B 0,C 180,E1 -26293.026,E2 -26293.026} C_VEL
LIN {X 0,Y 107.909,Z 407.041,A -85,B 0,C 180,E1 -26299.004,E2 -26299.004} C_VEL
LIN {X 0,Y 107.858,Z 407.045,A -85,B 0,C 180,E1 -26304.184,E2 -26304.184} C_VEL
LIN {X 0,Y 107.795,Z 407.055,A -85,B 0,C 180,E1 -26312.052,E2 -26312.052} C_VEL
LIN {X 0,Y 107.747,Z 407.063,A -85,B 0,C 180,E1 -26318.49,E2 -26318.49} C_VEL
LIN {X 0,Y 108.375,Z 407.097,A -85,B 0,C 180,E1 -26327.018,E2 -26327.018} C_VEL
LIN {X 0,Y 109.619,Z 411.589,A -85,B 0,C 180,E1 -26332.821,E2 -26332.821} C_VEL
LIN {X 0,Y 110.404,Z 413.99,A -85,B 0,C 180,E1 -26335.847,E2 -26335.847} C_VEL
LIN {X 0,Y 110.692,Z 415.503,A -85,B 0,C 180,E1 -26337.728,E2 -26337.728} C_VEL
LIN {X 0,Y 107.937,Z 423.975,A -85,B 0,C 180,E1 -26349.016,E2 -26349.016} C_VEL
LIN {X 0,Y 108.648,Z 429.132,A -85,B 0,C 180,E1 -26355.997,E2 -26355.997} C_VEL
LIN {X 0,Y 109.956,Z 431.502,A -85,B 0,C 180,E1 -26358.741,E2 -26358.741} C_VEL
LIN {X 0,Y 110.981,Z 444.27,A -85,B 0,C 180,E1 -26361.121,E2 -26361.121} C_VEL
LIN {X 0,Y 113.043,Z 456.991,A -85,B 0,C 180,E1 -26364.118,E2 -26364.118} C_VEL
LIN {X 0,Y 113.664,Z 461.377,A -85,B 0,C 180,E1 -26365.425,E2 -26365.425} C_VEL
LIN {X 0,Y 114.158,Z 470.936,A -85,B 0,C 180,E1 -26369.147,E2 -26369.147} C_VEL
LIN {X 0,Y 115.11,Z 479.754,A -85,B 0,C 180,E1 -26373.501,E2 -26373.501} C_VEL
LIN {X 0,Y 115.312,Z 481.697,A -85,B 0,C 180,E1 -26374.632,E2 -26374.632} C_VEL
LIN {X 0,Y 114.762,Z 484.644,A -85,B 0,C 180,E1 -26377.036,E2 -26377.036} C_VEL
LIN {X 0,Y 113.357,Z 489.775,A -85,B 0,C 180,E1 -26382.533,E2 -26382.533} C_VEL
LIN {X 0,Y 113.55,Z 495.298,A -85,B 0,C 180,E1 -26390.032,E2 -26390.032} C_VEL
LIN {X 0,Y 115.214,Z 498.576,A -85,B 0,C 180,E1 -26395.277,E2 -26395.277} C_VEL
LIN {X 0,Y 119.371,Z 502.167,A -85,B 0,C 180,E1 -26401.998,E2 -26401.998} C_VEL
LIN {X 0,Y 125.628,Z 504.831,A -85,B 0,C 180,E1 -26407.98,E2 -26407.98} C_VEL
LIN {X 0,Y 133.564,Z 506.649,A -85,B 0,C 180,E1 -26413.161,E2 -26413.161} C_VEL
LIN {X 0,Y 145.153,Z 507.736,A -85,B 0,C 180,E1 -26418.382,E2 -26418.382} C_VEL
LIN {X 0,Y 146.427,Z 507.772,A -85,B 0,C 180,E1 -26418.841,E2 -26418.841} C_VEL
LIN {X 0,Y 147.055,Z 507.534,A -85,B 0,C 180,E1 -26419.693,E2 -26419.693} C_VEL
LIN {X 0,Y 136.679,Z 503.632,A -85,B 0,C 180,E1 -26423.749,E2 -26423.749} C_VEL
LIN {X 0,Y 129.8,Z 499.662,A -85,B 0,C 180,E1 -26427.218,E2 -26427.218} C_VEL
LIN {X 0,Y 123.731,Z 494.782,A -85,B 0,C 180,E1 -26431.131,E2 -26431.131} C_VEL
LIN {X 0,Y 117.876,Z 487.658,A -85,B 0,C 180,E1 -26436.269,E2 -26436.269} C_VEL
LIN {X 0,Y 113.965,Z 480.316,A -85,B 0,C 180,E1 -26441.11,E2 -26441.11} C_VEL
LIN {X 0,Y 111.128,Z 469.918,A -85,B 0,C 180,E1 -26447.212,E2 -26447.212} C_VEL
LIN {X 0,Y 110.044,Z 460.052,A -85,B 0,C 180,E1 -26452.2,E2 -26452.2} C_VEL
LIN {X 0,Y 109.925,Z 447.786,A -85,B 0,C 180,E1 -26457.252,E2 -26457.252} C_VEL
LIN {X 0,Y 109.898,Z 436.301,A -85,B 0,C 180,E1 -26460.916,E2 -26460.916} C_VEL
LIN {X 0,Y 109.851,Z 429.186,A -85,B 0,C 180,E1 -26462.751,E2 -26462.751} C_VEL
LIN {X 0,Y 108.859,Z 422.514,A -85,B 0,C 180,E1 -26464.05,E2 -26464.05} C_VEL
LIN {X 0,Y 106.756,Z 419.321,A -85,B 0,C 180,E1 -26468.59,E2 -26468.59} C_VEL
LIN {X 0,Y 105.434,Z 417.32,A -85,B 0,C 180,E1 -26471.512,E2 -26471.512} C_VEL
LIN {X 0,Y 99.8,Z 410.106,A -85,B 0,C 180,E1 -26482.604,E2 -26482.604} C_VEL
LIN {X 0,Y 99.767,Z 408.785,A -85,B 0,C 180,E1 -26484.75,E2 -26484.75} C_VEL
LIN {X 0,Y 99.934,Z 408.036,A -85,B 0,C 180,E1 -26486.075,E2 -26486.075} C_VEL
LIN {X 0,Y 100.427,Z 407.979,A -85,B 0,C 180,E1 -26489.333,E2 -26489.333} C_VEL
LIN {X 0,Y 100.754,Z 407.92,A -85,B 0,C 180,E1 -26493.92,E2 -26493.92} C_VEL
LIN {X 0,Y 100.71,Z 407.939,A -85,B 0,C 180,E1 -26499.858,E2 -26499.858} C_VEL
LIN {X 0,Y 100.657,Z 407.945,A -85,B 0,C 180,E1 -26505.715,E2 -26505.715} C_VEL
LIN {X 0,Y 100.634,Z 407.942,A -85,B 0,C 180,E1 -26511.057,E2 -26511.057} C_VEL
LIN {X 0,Y 100.699,Z 407.94,A -85,B 0,C 180,E1 -26516.879,E2 -26516.879} C_VEL
LIN {X 0,Y 100.788,Z 407.93,A -85,B 0,C 180,E1 -26525.267,E2 -26525.267} C_VEL
LIN {X 0,Y 100.819,Z 407.921,A -85,B 0,C 180,E1 -26529.601,E2 -26529.601} C_VEL
LIN {X 0,Y 101.104,Z 407.883,A -85,B 0,C 180,E1 -26536.701,E2 -26536.701} C_VEL
LIN {X 0,Y 101.245,Z 407.874,A -85,B 0,C 180,E1 -26542.019,E2 -26542.019} C_VEL
LIN {X 0,Y 101.869,Z 407.797,A -85,B 0,C 180,E1 -26550,E2 -26550} C_VEL
LIN {X 0,Y 101.271,Z 407.871,A -85,B 0,C 180,E1 -26557.978,E2 -26557.978} C_VEL
LIN {X 0,Y 101.139,Z 407.879,A -85,B 0,C 180,E1 -26563.381,E2 -26563.381} C_VEL
LIN {X 0,Y 100.84,Z 407.918,A -85,B 0,C 180,E1 -26570.394,E2 -26570.394} C_VEL
LIN {X 0,Y 100.776,Z 407.931,A -85,B 0,C 180,E1 -26574.958,E2 -26574.958} C_VEL
LIN {X 0,Y 100.701,Z 407.94,A -85,B 0,C 180,E1 -26583.123,E2 -26583.123} C_VEL
LIN {X 0,Y 100.655,Z 407.942,A -85,B 0,C 180,E1 -26589.82,E2 -26589.82} C_VEL
LIN {X 0,Y 100.647,Z 407.943,A -85,B 0,C 180,E1 -26595.71,E2 -26595.71} C_VEL
LIN {X 0,Y 100.626,Z 407.951,A -85,B 0,C 180,E1 -26601.053,E2 -26601.053} C_VEL
LIN {X 0,Y 100.692,Z 407.936,A -85,B 0,C 180,E1 -26606.883,E2 -26606.883} C_VEL
LIN {X 0,Y 100.787,Z 407.924,A -85,B 0,C 180,E1 -26615.267,E2 -26615.267} C_VEL
LIN {X 0,Y 100.821,Z 407.925,A -85,B 0,C 180,E1 -26619.602,E2 -26619.602} C_VEL
LIN {X 0,Y 101.2,Z 407.879,A -85,B 0,C 180,E1 -26627.975,E2 -26627.975} C_VEL
LIN {X 0,Y 101.281,Z 407.861,A -85,B 0,C 180,E1 -26632.022,E2 -26632.022} C_VEL
LIN {X 0,Y 101.873,Z 407.788,A -85,B 0,C 180,E1 -26640,E2 -26640} C_VEL
LIN {X 0,Y 101.281,Z 407.862,A -85,B 0,C 180,E1 -26647.977,E2 -26647.977} C_VEL
LIN {X 0,Y 101.13,Z 407.887,A -85,B 0,C 180,E1 -26653.363,E2 -26653.363} C_VEL
LIN {X 0,Y 100.819,Z 407.927,A -85,B 0,C 180,E1 -26660.398,E2 -26660.398} C_VEL
LIN {X 0,Y 100.775,Z 407.926,A -85,B 0,C 180,E1 -26664.958,E2 -26664.958} C_VEL
LIN {X 0,Y 100.702,Z 407.936,A -85,B 0,C 180,E1 -26673.125,E2 -26673.125} C_VEL
LIN {X 0,Y 100.716,Z 407.938,A -85,B 0,C 180,E1 -26679.863,E2 -26679.863} C_VEL
LIN {X 0,Y 101.399,Z 407.961,A -85,B 0,C 180,E1 -26687.821,E2 -26687.821} C_VEL
LIN {X 0,Y 103.012,Z 413.138,A -85,B 0,C 180,E1 -26694.955,E2 -26694.955} C_VEL
LIN {X 0,Y 103.455,Z 414.723,A -85,B 0,C 180,E1 -26697.08,E2 -26697.08} C_VEL
LIN {X 0,Y 103.066,Z 416.295,A -85,B 0,C 180,E1 -26699.242,E2 -26699.242} C_VEL
LIN {X 0,Y 101.479,Z 427.642,A -85,B 0,C 180,E1 -26715.832,E2 -26715.832} C_VEL
LIN {X 0,Y 103.472,Z 430.866,A -85,B 0,C 180,E1 -26720.224,E2 -26720.224} C_VEL
LIN {X 0,Y 104.821,Z 444.517,A -85,B 0,C 180,E1 -26723.018,E2 -26723.018} C_VEL
LIN {X 0,Y 106.728,Z 455.26,A -85,B 0,C 180,E1 -26725.676,E2 -26725.676} C_VEL
LIN {X 0,Y 107.466,Z 458.881,A -85,B 0,C 180,E1 -26726.72,E2 -26726.72} C_VEL
LIN {X 0,Y 108.212,Z 469.147,A -85,B 0,C 180,E1 -26730.931,E2 -26730.931} C_VEL
LIN {X 0,Y 109.248,Z 477.68,A -85,B 0,C 180,E1 -26735.295,E2 -26735.295} C_VEL
LIN {X 0,Y 109.299,Z 479.243,A -85,B 0,C 180,E1 -26736.34,E2 -26736.34} C_VEL
LIN {X 0,Y 108.215,Z 483.038,A -85,B 0,C 180,E1 -26739.965,E2 -26739.965} C_VEL
LIN {X 0,Y 107.491,Z 490.354,A -85,B 0,C 180,E1 -26749.082,E2 -26749.082} C_VEL
LIN {X 0,Y 109.583,Z 495.269,A -85,B 0,C 180,E1 -26756.676,E2 -26756.676} C_VEL
LIN {X 0,Y 113.959,Z 499.179,A -85,B 0,C 180,E1 -26763.714,E2 -26763.714} C_VEL
LIN {X 0,Y 120.482,Z 502.253,A -85,B 0,C 180,E1 -26769.916,E2 -26769.916} C_VEL
LIN {X 0,Y 128.73,Z 504.431,A -85,B 0,C 180,E1 -26775.214,E2 -26775.214} C_VEL
LIN {X 0,Y 136.331,Z 505.625,A -85,B 0,C 180,E1 -26778.771,E2 -26778.771} C_VEL
LIN {X 0,Y 135.662,Z 504.952,A -85,B 0,C 180,E1 -26779.993,E2 -26779.993} C_VEL
LIN {X 0,Y 126.216,Z 499.937,A -85,B 0,C 180,E1 -26784.221,E2 -26784.221} C_VEL
LIN {X 0,Y 119.638,Z 494.839,A -85,B 0,C 180,E1 -26788.083,E2 -26788.083} C_VEL
LIN {X 0,Y 113.189,Z 487.695,A -85,B 0,C 180,E1 -26793.246,E2 -26793.246} C_VEL
LIN {X 0,Y 108.217,Z 478.866,A -85,B 0,C 180,E1 -26799.073,E2 -26799.073} C_VEL
LIN {X 0,Y 105.401,Z 469.846,A -85,B 0,C 180,E1 -26804.531,E2 -26804.531} C_VEL
LIN {X 0,Y 103.926,Z 458.964,A -85,B 0,C 180,E1 -26810.267,E2 -26810.267} C_VEL
LIN {X 0,Y 103.537,Z 447.876,A -85,B 0,C 180,E1 -26815.133,E2 -26815.133} C_VEL
LIN {X 0,Y 103.489,Z 439.592,A -85,B 0,C 180,E1 -26818.054,E2 -26818.054} C_VEL
LIN {X 0,Y 103.427,Z 429.385,A -85,B 0,C 180,E1 -26820.974,E2 -26820.974} C_VEL
LIN {X 0,Y 102.497,Z 422.897,A -85,B 0,C 180,E1 -26822.334,E2 -26822.334} C_VEL
LIN {X 0,Y 99.703,Z 419.052,A -85,B 0,C 180,E1 -26828.105,E2 -26828.105} C_VEL
LIN {X 0,Y 99.312,Z 411.261,A -85,B 0,C 180,E1 -26840.723,E2 -26840.723} C_VEL
LIN {X 0,Y 99.767,Z 408.785,A -85,B 0,C 180,E1 -26844.75,E2 -26844.75} C_VEL
LIN {X 0,Y 99.675,Z 408.126,A -85,B 0,C 180,E1 -26846.913,E2 -26846.913} C_VEL
LIN {X 0,Y 99.068,Z 408.148,A -85,B 0,C 180,E1 -26849.127,E2 -26849.127} C_VEL
LIN {X 0,Y 97.007,Z 408.387,A -85,B 0,C 180,E1 -26853.616,E2 -26853.616} C_VEL
LIN {X 0,Y 93.904,Z 408.816,A -85,B 0,C 180,E1 -26860.857,E2 -26860.857} C_VEL
LIN {X 0,Y 93.511,Z 408.824,A -85,B 0,C 180,E1 -26863.381,E2 -26863.381} C_VEL
LIN {X 0,Y 93.541,Z 408.831,A -85,B 0,C 180,E1 -26868.706,E2 -26868.706} C_VEL
LIN {X 0,Y 93.595,Z 408.826,A -85,B 0,C 180,E1 -26875.69,E2 -26875.69} C_VEL
LIN {X 0,Y 93.671,Z 408.817,A -85,B 0,C 180,E1 -26884.205,E2 -26884.205} C_VEL
LIN {X 0,Y 93.695,Z 408.807,A -85,B 0,C 180,E1 -26887.972,E2 -26887.972} C_VEL
LIN {X 0,Y 94.024,Z 408.765,A -85,B 0,C 180,E1 -26896.341,E2 -26896.341} C_VEL
LIN {X 0,Y 94.178,Z 408.754,A -85,B 0,C 180,E1 -26901.416,E2 -26901.416} C_VEL
LIN {X 0,Y 94.795,Z 408.678,A -85,B 0,C 180,E1 -26910,E2 -26910} C_VEL
LIN {X 0,Y 94.206,Z 408.75,A -85,B 0,C 180,E1 -26918.581,E2 -26918.581} C_VEL
LIN {X 0,Y 94.055,Z 408.762,A -85,B 0,C 180,E1 -26923.736,E2 -26923.736} C_VEL
LIN {X 0,Y 93.707,Z 408.805,A -85,B 0,C 180,E1 -26932.024,E2 -26932.024} C_VEL
LIN {X 0,Y 93.625,Z 408.822,A -85,B 0,C 180,E1 -26936.769,E2 -26936.769} C_VEL
LIN {X 0,Y 93.6,Z 408.826,A -85,B 0,C 180,E1 -26944.315,E2 -26944.315} C_VEL
LIN {X 0,Y 93.538,Z 408.833,A -85,B 0,C 180,E1 -26952.548,E2 -26952.548} C_VEL
LIN {X 0,Y 93.534,Z 408.829,A -85,B 0,C 180,E1 -26958.71,E2 -26958.71} C_VEL
LIN {X 0,Y 93.588,Z 408.819,A -85,B 0,C 180,E1 -26965.694,E2 -26965.694} C_VEL
LIN {X 0,Y 93.67,Z 408.809,A -85,B 0,C 180,E1 -26974.205,E2 -26974.205} C_VEL
LIN {X 0,Y 93.696,Z 408.813,A -85,B 0,C 180,E1 -26977.973,E2 -26977.973} C_VEL
LIN {X 0,Y 94.099,Z 408.764,A -85,B 0,C 180,E1 -26987.052,E2 -26987.052} C_VEL
LIN {X 0,Y 94.213,Z 408.741,A -85,B 0,C 180,E1 -26991.419,E2 -26991.419} C_VEL
LIN {X 0,Y 94.799,Z 408.668,A -85,B 0,C 180,E1 -27000,E2 -27000} C_VEL
LIN {X 0,Y 94.213,Z 408.742,A -85,B 0,C 180,E1 -27008.58,E2 -27008.58} C_VEL
LIN {X 0,Y 94.048,Z 408.77,A -85,B 0,C 180,E1 -27013.721,E2 -27013.721} C_VEL
LIN {X 0,Y 93.695,Z 408.814,A -85,B 0,C 180,E1 -27022.027,E2 -27022.027} C_VEL
LIN {X 0,Y 93.623,Z 408.817,A -85,B 0,C 180,E1 -27026.769,E2 -27026.769} C_VEL
LIN {X 0,Y 93.606,Z 408.817,A -85,B 0,C 180,E1 -27034.322,E2 -27034.322} C_VEL
LIN {X 0,Y 93.78,Z 408.795,A -85,B 0,C 180,E1 -27042.413,E2 -27042.413} C_VEL
LIN {X 0,Y 94.494,Z 408.833,A -85,B 0,C 180,E1 -27048.855,E2 -27048.855} C_VEL
LIN {X 0,Y 96.241,Z 414.217,A -85,B 0,C 180,E1 -27056.792,E2 -27056.792} C_VEL
LIN {X 0,Y 95.93,Z 415.796,A -85,B 0,C 180,E1 -27059.148,E2 -27059.148} C_VEL
LIN {X 0,Y 94.337,Z 426.103,A -85,B 0,C 180,E1 -27075.577,E2 -27075.577} C_VEL
LIN {X 0,Y 95.569,Z 428.597,A -85,B 0,C 180,E1 -27079.406,E2 -27079.406} C_VEL
LIN {X 0,Y 97.301,Z 430.834,A -85,B 0,C 180,E1 -27082.293,E2 -27082.293} C_VEL
LIN {X 0,Y 98.758,Z 443.863,A -85,B 0,C 180,E1 -27085.064,E2 -27085.064} C_VEL
LIN {X 0,Y 100.996,Z 455.175,A -85,B 0,C 180,E1 -27088.006,E2 -27088.006} C_VEL
LIN {X 0,Y 101.523,Z 458.247,A -85,B 0,C 180,E1 -27089.009,E2 -27089.009} C_VEL
LIN {X 0,Y 102.393,Z 467.395,A -85,B 0,C 180,E1 -27092.951,E2 -27092.951} C_VEL
LIN {X 0,Y 103.432,Z 474.763,A -85,B 0,C 180,E1 -27096.829,E2 -27096.829} C_VEL
LIN {X 0,Y 103.405,Z 476.095,A -85,B 0,C 180,E1 -27097.813,E2 -27097.813} C_VEL
LIN {X 0,Y 101.834,Z 482.54,A -85,B 0,C 180,E1 -27104.94,E2 -27104.94} C_VEL
LIN {X 0,Y 102.198,Z 487.898,A -85,B 0,C 180,E1 -27112.224,E2 -27112.224} C_VEL
LIN {X 0,Y 104.487,Z 492.28,A -85,B 0,C 180,E1 -27119.025,E2 -27119.025} C_VEL
LIN {X 0,Y 111.911,Z 497.785,A -85,B 0,C 180,E1 -27128.903,E2 -27128.903} C_VEL
LIN {X 0,Y 122.482,Z 501.533,A -85,B 0,C 180,E1 -27136.484,E2 -27136.484} C_VEL
LIN {X 0,Y 125.709,Z 502.306,A -85,B 0,C 180,E1 -27138.186,E2 -27138.186} C_VEL
LIN {X 0,Y 126.547,Z 502.134,A -85,B 0,C 180,E1 -27139.468,E2 -27139.468} C_VEL
LIN {X 0,Y 118.231,Z 496.728,A -85,B 0,C 180,E1 -27143.528,E2 -27143.528} C_VEL
LIN {X 0,Y 110.792,Z 489.779,A -85,B 0,C 180,E1 -27148.444,E2 -27148.444} C_VEL
LIN {X 0,Y 104.783,Z 481.423,A -85,B 0,C 180,E1 -27154.153,E2 -27154.153} C_VEL
LIN {X 0,Y 100.458,Z 471.191,A -85,B 0,C 180,E1 -27160.591,E2 -27160.591} C_VEL
LIN {X 0,Y 98.525,Z 462.621,A -85,B 0,C 180,E1 -27165.543,E2 -27165.543} C_VEL
LIN {X 0,Y 97.558,Z 452.311,A -85,B 0,C 180,E1 -27170.672,E2 -27170.672} C_VEL
LIN {X 0,Y 97.342,Z 441.081,A -85,B 0,C 180,E1 -27175.341,E2 -27175.341} C_VEL
LIN {X 0,Y 97.116,Z 429.58,A -85,B 0,C 180,E1 -27178.964,E2 -27178.964} C_VEL
LIN {X 0,Y 96.235,Z 423.236,A -85,B 0,C 180,E1 -27180.393,E2 -27180.393} C_VEL
LIN {X 0,Y 93.023,Z 419.385,A -85,B 0,C 180,E1 -27186.47,E2 -27186.47} C_VEL
LIN {X 0,Y 92.37,Z 410.236,A -85,B 0,C 180,E1 -27202.361,E2 -27202.361} C_VEL
LIN {X 0,Y 92.711,Z 408.934,A -85,B 0,C 180,E1 -27205.06,E2 -27205.06} C_VEL
LIN {X 0,Y 93.021,Z 408.898,A -85,B 0,C 180,E1 -27206.957,E2 -27206.957} C_VEL
LIN {X 0,Y 93.53,Z 408.829,A -85,B 0,C 180,E1 -27211.736,E2 -27211.736} C_VEL
LIN {X 0,Y 93.67,Z 408.804,A -85,B 0,C 180,E1 -27214.377,E2 -27214.377} C_VEL
LIN {X 0,Y 93.565,Z 408.823,A -85,B 0,C 180,E1 -27222.535,E2 -27222.535} C_VEL
LIN {X 0,Y 93.511,Z 408.824,A -85,B 0,C 180,E1 -27223.381,E2 -27223.381} C_VEL
LIN {X 0,Y 92.761,Z 408.931,A -85,B 0,C 180,E1 -27226.985,E2 -27226.985} C_VEL
LIN {X 0,Y 91.244,Z 409.118,A -85,B 0,C 180,E1 -27230.565,E2 -27230.565} C_VEL
LIN {X 0,Y 86.947,Z 409.663,A -85,B 0,C 180,E1 -27240.591,E2 -27240.591} C_VEL
LIN {X 0,Y 86.586,Z 409.699,A -85,B 0,C 180,E1 -27243.257,E2 -27243.257} C_VEL
LIN {X 0,Y 86.648,Z 409.69,A -85,B 0,C 180,E1 -27251.068,E2 -27251.068} C_VEL
LIN {X 0,Y 86.933,Z 409.65,A -85,B 0,C 180,E1 -27255.964,E2 -27255.964} C_VEL
LIN {X 0,Y 87.087,Z 409.637,A -85,B 0,C 180,E1 -27260.711,E2 -27260.711} C_VEL
LIN {X 0,Y 87.721,Z 409.559,A -85,B 0,C 180,E1 -27270,E2 -27270} C_VEL
LIN {X 0,Y 87.115,Z 409.634,A -85,B 0,C 180,E1 -27279.285,E2 -27279.285} C_VEL
LIN {X 0,Y 86.976,Z 409.645,A -85,B 0,C 180,E1 -27284.149,E2 -27284.149} C_VEL
LIN {X 0,Y 86.677,Z 409.687,A -85,B 0,C 180,E1 -27288.925,E2 -27288.925} C_VEL
LIN {X 0,Y 86.587,Z 409.699,A -85,B 0,C 180,E1 -27296.766,E2 -27296.766} C_VEL
LIN {X 0,Y 86.518,Z 409.706,A -85,B 0,C 180,E1 -27305.676,E2 -27305.676} C_VEL
LIN {X 0,Y 86.48,Z 409.713,A -85,B 0,C 180,E1 -27312.995,E2 -27312.995} C_VEL
LIN {X 0,Y 86.456,Z 409.713,A -85,B 0,C 180,E1 -27319.434,E2 -27319.434} C_VEL
LIN {X 0,Y 86.531,Z 409.698,A -85,B 0,C 180,E1 -27325.351,E2 -27325.351} C_VEL
LIN {X 0,Y 86.585,Z 409.693,A -85,B 0,C 180,E1 -27333.234,E2 -27333.234} C_VEL
LIN {X 0,Y 86.667,Z 409.685,A -85,B 0,C 180,E1 -27341.072,E2 -27341.072} C_VEL
LIN {X 0,Y 86.97,Z 409.651,A -85,B 0,C 180,E1 -27345.97,E2 -27345.97} C_VEL
LIN {X 0,Y 87.119,Z 409.625,A -85,B 0,C 180,E1 -27350.715,E2 -27350.715} C_VEL
LIN {X 0,Y 87.727,Z 409.549,A -85,B 0,C 180,E1 -27360,E2 -27360} C_VEL
LIN {X 0,Y 87.119,Z 409.626,A -85,B 0,C 180,E1 -27369.284,E2 -27369.284} C_VEL
LIN {X 0,Y 86.951,Z 409.653,A -85,B 0,C 180,E1 -27374.087,E2 -27374.087} C_VEL
LIN {X 0,Y 86.665,Z 409.686,A -85,B 0,C 180,E1 -27378.927,E2 -27378.927} C_VEL
LIN {X 0,Y 86.585,Z 409.693,A -85,B 0,C 180,E1 -27386.766,E2 -27386.766} C_VEL
LIN {X 0,Y 86.533,Z 409.7,A -85,B 0,C 180,E1 -27395.692,E2 -27395.692} C_VEL
LIN {X 0,Y 86.773,Z 409.667,A -85,B 0,C 180,E1 -27403.203,E2 -27403.203} C_VEL
LIN {X 0,Y 87.603,Z 409.662,A -85,B 0,C 180,E1 -27410.074,E2 -27410.074} C_VEL
LIN {X 0,Y 88.984,Z 413.647,A -85,B 0,C 180,E1 -27416.437,E2 -27416.437} C_VEL
LIN {X 0,Y 88.797,Z 415.253,A -85,B 0,C 180,E1 -27419.042,E2 -27419.042} C_VEL
LIN {X 0,Y 87.371,Z 424.98,A -85,B 0,C 180,E1 -27436.036,E2 -27436.036} C_VEL
LIN {X 0,Y 88.943,Z 427.892,A -85,B 0,C 180,E1 -27440.908,E2 -27440.908} C_VEL
LIN {X 0,Y 91.227,Z 430.451,A -85,B 0,C 180,E1 -27444.51,E2 -27444.51} C_VEL
LIN {X 0,Y 92.781,Z 442.85,A -85,B 0,C 180,E1 -27447.287,E2 -27447.287} C_VEL
LIN {X 0,Y 95.37,Z 454.795,A -85,B 0,C 180,E1 -27450.528,E2 -27450.528} C_VEL
LIN {X 0,Y 96.205,Z 461.18,A -85,B 0,C 180,E1 -27453.141,E2 -27453.141} C_VEL
LIN {X 0,Y 97.406,Z 469.338,A -85,B 0,C 180,E1 -27457.254,E2 -27457.254} C_VEL
LIN {X 0,Y 97.771,Z 472.403,A -85,B 0,C 180,E1 -27459.2,E2 -27459.2} C_VEL
LIN {X 0,Y 96.313,Z 479.171,A -85,B 0,C 180,E1 -27466.971,E2 -27466.971} C_VEL
LIN {X 0,Y 97.975,Z 486.694,A -85,B 0,C 180,E1 -27477.792,E2 -27477.792} C_VEL
LIN {X 0,Y 103.76,Z 492.51,A -85,B 0,C 180,E1 -27487.561,E2 -27487.561} C_VEL
LIN {X 0,Y 110.943,Z 496.226,A -85,B 0,C 180,E1 -27494.173,E2 -27494.173} C_VEL
LIN {X 0,Y 115.164,Z 497.812,A -85,B 0,C 180,E1 -27497.081,E2 -27497.081} C_VEL
LIN {X 0,Y 117.631,Z 498.415,A -85,B 0,C 180,E1 -27498.913,E2 -27498.913} C_VEL
LIN {X 0,Y 108.161,Z 490.7,A -85,B 0,C 180,E1 -27504.212,E2 -27504.212} C_VEL
LIN {X 0,Y 101.348,Z 482.384,A -85,B 0,C 180,E1 -27509.818,E2 -27509.818} C_VEL
LIN {X 0,Y 96.666,Z 473.98,A -85,B 0,C 180,E1 -27515.289,E2 -27515.289} C_VEL
LIN {X 0,Y 93.535,Z 463.98,A -85,B 0,C 180,E1 -27521.378,E2 -27521.378} C_VEL
LIN {X 0,Y 91.867,Z 453.133,A -85,B 0,C 180,E1 -27527.295,E2 -27527.295} C_VEL
LIN {X 0,Y 91.354,Z 440.719,A -85,B 0,C 180,E1 -27532.819,E2 -27532.819} C_VEL
LIN {X 0,Y 90.977,Z 428.329,A -85,B 0,C 180,E1 -27536.956,E2 -27536.956} C_VEL
LIN {X 0,Y 90.227,Z 423.624,A -85,B 0,C 180,E1 -27538.047,E2 -27538.047} C_VEL
LIN {X 0,Y 86.412,Z 419.629,A -85,B 0,C 180,E1 -27544.666,E2 -27544.666} C_VEL
LIN {X 0,Y 85.33,Z 409.856,A -85,B 0,C 180,E1 -27563.031,E2 -27563.031} C_VEL
LIN {X 0,Y 85.739,Z 409.802,A -85,B 0,C 180,E1 -27565.62,E2 -27565.62} C_VEL
LIN {X 0,Y 86.133,Z 409.759,A -85,B 0,C 180,E1 -27569.313,E2 -27569.313} C_VEL
LIN {X 0,Y 86.582,Z 409.694,A -85,B 0,C 180,E1 -27575.735,E2 -27575.735} C_VEL
LIN {X 0,Y 86.489,Z 409.703,A -85,B 0,C 180,E1 -27583.235,E2 -27583.235} C_VEL
LIN {X 0,Y 86.462,Z 409.712,A -85,B 0,C 180,E1 -27589.437,E2 -27589.437} C_VEL
LIN {X 0,Y 86.538,Z 409.705,A -85,B 0,C 180,E1 -27595.354,E2 -27595.354} C_VEL
LIN {X 0,Y 86.586,Z 409.699,A -85,B 0,C 180,E1 -27603.257,E2 -27603.257} C_VEL
LIN {X 0,Y 85.826,Z 409.79,A -85,B 0,C 180,E1 -27607.144,E2 -27607.144} C_VEL
LIN {X 0,Y 84.252,Z 409.989,A -85,B 0,C 180,E1 -27611.009,E2 -27611.009} C_VEL
LIN {X 0,Y 80.186,Z 410.497,A -85,B 0,C 180,E1 -27621.927,E2 -27621.927} C_VEL
LIN {X 0,Y 80.11,Z 410.498,A -85,B 0,C 180,E1 -27624.821,E2 -27624.821} C_VEL
LIN {X 0,Y 80.648,Z 410.44,A -85,B 0,C 180,E1 -27630,E2 -27630} C_VEL
LIN {X 0,Y 79.999,Z 410.518,A -85,B 0,C 180,E1 -27640.119,E2 -27640.119} C_VEL
LIN {X 0,Y 79.817,Z 410.54,A -85,B 0,C 180,E1 -27645.316,E2 -27645.316} C_VEL
LIN {X 0,Y 79.533,Z 410.57,A -85,B 0,C 180,E1 -27650.699,E2 -27650.699} C_VEL
LIN {X 0,Y 79.485,Z 410.581,A -85,B 0,C 180,E1 -27657.846,E2 -27657.846} C_VEL
LIN {X 0,Y 79.386,Z 410.593,A -85,B 0,C 180,E1 -27662.085,E2 -27662.085} C_VEL
LIN {X 0,Y 79.373,Z 410.589,A -85,B 0,C 180,E1 -27668.302,E2 -27668.302} C_VEL
LIN {X 0,Y 79.387,Z 410.592,A -85,B 0,C 180,E1 -27675.091,E2 -27675.091} C_VEL
LIN {X 0,Y 79.386,Z 410.595,A -85,B 0,C 180,E1 -27682.822,E2 -27682.822} C_VEL
LIN {X 0,Y 79.378,Z 410.595,A -85,B 0,C 180,E1 -27687.911,E2 -27687.911} C_VEL
LIN {X 0,Y 79.526,Z 410.571,A -85,B 0,C 180,E1 -27693.776,E2 -27693.776} C_VEL
LIN {X 0,Y 79.526,Z 410.578,A -85,B 0,C 180,E1 -27699.298,E2 -27699.298} C_VEL
LIN {X 0,Y 79.842,Z 410.538,A -85,B 0,C 180,E1 -27705.525,E2 -27705.525} C_VEL
LIN {X 0,Y 80.001,Z 410.514,A -85,B 0,C 180,E1 -27709.88,E2 -27709.88} C_VEL
LIN {X 0,Y 80.655,Z 410.43,A -85,B 0,C 180,E1 -27720,E2 -27720} C_VEL
LIN {X 0,Y 80.001,Z 410.514,A -85,B 0,C 180,E1 -27730.119,E2 -27730.119} C_VEL
LIN {X 0,Y 79.766,Z 410.545,A -85,B 0,C 180,E1 -27735.326,E2 -27735.326} C_VEL
LIN {X 0,Y 79.524,Z 410.579,A -85,B 0,C 180,E1 -27740.701,E2 -27740.701} C_VEL
LIN {X 0,Y 79.484,Z 410.581,A -85,B 0,C 180,E1 -27747.846,E2 -27747.846} C_VEL
LIN {X 0,Y 79.463,Z 410.585,A -85,B 0,C 180,E1 -27757.251,E2 -27757.251} C_VEL
LIN {X 0,Y 80.227,Z 410.492,A -85,B 0,C 180,E1 -27768.158,E2 -27768.158} C_VEL
LIN {X 0,Y 80.741,Z 410.473,A -85,B 0,C 180,E1 -27771.572,E2 -27771.572} C_VEL
LIN {X 0,Y 81.706,Z 413.017,A -85,B 0,C 180,E1 -27776.006,E2 -27776.006} C_VEL
LIN {X 0,Y 81.472,Z 415.041,A -85,B 0,C 180,E1 -27779.612,E2 -27779.612} C_VEL
LIN {X 0,Y 80.594,Z 424.287,A -85,B 0,C 180,E1 -27797.454,E2 -27797.454} C_VEL
LIN {X 0,Y 82.4,Z 427.148,A -85,B 0,C 180,E1 -27802.65,E2 -27802.65} C_VEL
LIN {X 0,Y 85.395,Z 429.973,A -85,B 0,C 180,E1 -27807.115,E2 -27807.115} C_VEL
LIN {X 0,Y 87.383,Z 443.202,A -85,B 0,C 180,E1 -27810.288,E2 -27810.288} C_VEL
LIN {X 0,Y 89.981,Z 453.93,A -85,B 0,C 180,E1 -27813.359,E2 -27813.359} C_VEL
LIN {X 0,Y 91.055,Z 461.251,A -85,B 0,C 180,E1 -27816.649,E2 -27816.649} C_VEL
LIN {X 0,Y 92.144,Z 467.274,A -85,B 0,C 180,E1 -27819.882,E2 -27819.882} C_VEL
LIN {X 0,Y 92.23,Z 468.82,A -85,B 0,C 180,E1 -27820.982,E2 -27820.982} C_VEL
LIN {X 0,Y 91.124,Z 476.445,A -85,B 0,C 180,E1 -27830.397,E2 -27830.397} C_VEL
LIN {X 0,Y 92.932,Z 482.546,A -85,B 0,C 180,E1 -27839.444,E2 -27839.444} C_VEL
LIN {X 0,Y 97.157,Z 487.4,A -85,B 0,C 180,E1 -27847.279,E2 -27847.279} C_VEL
LIN {X 0,Y 106.551,Z 492.866,A -85,B 0,C 180,E1 -27856.515,E2 -27856.515} C_VEL
LIN {X 0,Y 107.746,Z 493.368,A -85,B 0,C 180,E1 -27857.375,E2 -27857.375} C_VEL
LIN {X 0,Y 108.499,Z 493.424,A -85,B 0,C 180,E1 -27858.546,E2 -27858.546} C_VEL
LIN {X 0,Y 99.518,Z 484.531,A -85,B 0,C 180,E1 -27864.365,E2 -27864.365} C_VEL
LIN {X 0,Y 93.107,Z 474.907,A -85,B 0,C 180,E1 -27870.617,E2 -27870.617} C_VEL
LIN {X 0,Y 89.054,Z 465.23,A -85,B 0,C 180,E1 -27876.76,E2 -27876.76} C_VEL
LIN {X 0,Y 86.624,Z 453.538,A -85,B 0,C 180,E1 -27883.503,E2 -27883.503} C_VEL
LIN {X 0,Y 85.562,Z 441.592,A -85,B 0,C 180,E1 -27889.35,E2 -27889.35} C_VEL
LIN {X 0,Y 85.176,Z 432.513,A -85,B 0,C 180,E1 -27892.84,E2 -27892.84} C_VEL
LIN {X 0,Y 84.932,Z 426.602,A -85,B 0,C 180,E1 -27894.708,E2 -27894.708} C_VEL
LIN {X 0,Y 84.394,Z 423.965,A -85,B 0,C 180,E1 -27895.373,E2 -27895.373} C_VEL
LIN {X 0,Y 79.936,Z 419.855,A -85,B 0,C 180,E1 -27902.52,E2 -27902.52} C_VEL
LIN {X 0,Y 77.709,Z 414.582,A -85,B 0,C 180,E1 -27913.068,E2 -27913.068} C_VEL
LIN {X 0,Y 78.034,Z 410.767,A -85,B 0,C 180,E1 -27921.116,E2 -27921.116} C_VEL
LIN {X 0,Y 78.79,Z 410.669,A -85,B 0,C 180,E1 -27926.873,E2 -27926.873} C_VEL
LIN {X 0,Y 79.256,Z 410.604,A -85,B 0,C 180,E1 -27932.145,E2 -27932.145} C_VEL
LIN {X 0,Y 79.45,Z 410.588,A -85,B 0,C 180,E1 -27938.259,E2 -27938.259} C_VEL
LIN {X 0,Y 79.414,Z 410.59,A -85,B 0,C 180,E1 -27945.072,E2 -27945.072} C_VEL
LIN {X 0,Y 79.391,Z 410.589,A -85,B 0,C 180,E1 -27952.819,E2 -27952.819} C_VEL
LIN {X 0,Y 79.383,Z 410.593,A -85,B 0,C 180,E1 -27957.913,E2 -27957.913} C_VEL
LIN {X 0,Y 79.527,Z 410.578,A -85,B 0,C 180,E1 -27963.777,E2 -27963.777} C_VEL
LIN {X 0,Y 79.515,Z 410.573,A -85,B 0,C 180,E1 -27969.295,E2 -27969.295} C_VEL
LIN {X 0,Y 79.826,Z 410.536,A -85,B 0,C 180,E1 -27975.572,E2 -27975.572} C_VEL
LIN {X 0,Y 79.97,Z 410.522,A -85,B 0,C 180,E1 -27979.876,E2 -27979.876} C_VEL
LIN {X 0,Y 80.11,Z 410.498,A -85,B 0,C 180,E1 -27984.821,E2 -27984.821} C_VEL
LIN {X 0,Y 79.976,Z 410.529,A -85,B 0,C 180,E1 -27987.618,E2 -27987.618} C_VEL
LIN {X 0,Y 78.726,Z 410.701,A -85,B 0,C 180,E1 -27991.785,E2 -27991.785} C_VEL
LIN {X 0,Y 76.798,Z 410.947,A -85,B 0,C 180,E1 -27995.946,E2 -27995.946} C_VEL
LIN {X 0,Y 73.029,Z 411.394,A -85,B 0,C 180,E1 -28005.009,E2 -28005.009} C_VEL
LIN {X 0,Y 72.496,Z 411.445,A -85,B 0,C 180,E1 -28008.237,E2 -28008.237} C_VEL
LIN {X 0,Y 72.406,Z 411.46,A -85,B 0,C 180,E1 -28012.846,E2 -28012.846} C_VEL
LIN {X 0,Y 72.378,Z 411.462,A -85,B 0,C 180,E1 -28019.082,E2 -28019.082} C_VEL
LIN {X 0,Y 72.301,Z 411.477,A -85,B 0,C 180,E1 -28025.678,E2 -28025.678} C_VEL
LIN {X 0,Y 72.248,Z 411.486,A -85,B 0,C 180,E1 -28032.916,E2 -28032.916} C_VEL
LIN {X 0,Y 72.294,Z 411.48,A -85,B 0,C 180,E1 -28041.052,E2 -28041.052} C_VEL
LIN {X 0,Y 72.294,Z 411.473,A -85,B 0,C 180,E1 -28044.317,E2 -28044.317} C_VEL
LIN {X 0,Y 72.375,Z 411.469,A -85,B 0,C 180,E1 -28050.952,E2 -28050.952} C_VEL
LIN {X 0,Y 72.401,Z 411.465,A -85,B 0,C 180,E1 -28057.152,E2 -28057.152} C_VEL
LIN {X 0,Y 72.758,Z 411.418,A -85,B 0,C 180,E1 -28065.002,E2 -28065.002} C_VEL
LIN {X 0,Y 72.886,Z 411.404,A -85,B 0,C 180,E1 -28068.88,E2 -28068.88} C_VEL
LIN {X 0,Y 73.582,Z 411.311,A -85,B 0,C 180,E1 -28080,E2 -28080} C_VEL
LIN {X 0,Y 72.886,Z 411.404,A -85,B 0,C 180,E1 -28091.119,E2 -28091.119} C_VEL
LIN {X 0,Y 72.587,Z 411.434,A -85,B 0,C 180,E1 -28096.885,E2 -28096.885} C_VEL
LIN {X 0,Y 72.4,Z 411.465,A -85,B 0,C 180,E1 -28102.848,E2 -28102.848} C_VEL
LIN {X 0,Y 72.377,Z 411.469,A -85,B 0,C 180,E1 -28109.082,E2 -28109.082} C_VEL
LIN {X 0,Y 72.418,Z 411.464,A -85,B 0,C 180,E1 -28119.07,E2 -28119.07} C_VEL
LIN {X 0,Y 73.418,Z 411.341,A -85,B 0,C 180,E1 -28129.978,E2 -28129.978} C_VEL
LIN {X 0,Y 74.01,Z 411.441,A -85,B 0,C 180,E1 -28133.767,E2 -28133.767} C_VEL
LIN {X 0,Y 74.605,Z 413.633,A -85,B 0,C 180,E1 -28137.976,E2 -28137.976} C_VEL
LIN {X 0,Y 73.851,Z 423.498,A -85,B 0,C 180,E1 -28159.028,E2 -28159.028} C_VEL
LIN {X 0,Y 77.406,Z 427.712,A -85,B 0,C 180,E1 -28167.117,E2 -28167.117} C_VEL
LIN {X 0,Y 79.85,Z 429.59,A -85,B 0,C 180,E1 -28170.158,E2 -28170.158} C_VEL
LIN {X 0,Y 82.268,Z 443.4,A -85,B 0,C 180,E1 -28173.674,E2 -28173.674} C_VEL
LIN {X 0,Y 84.853,Z 453.158,A -85,B 0,C 180,E1 -28176.598,E2 -28176.598} C_VEL
LIN {X 0,Y 86.571,Z 462.541,A -85,B 0,C 180,E1 -28181.295,E2 -28181.295} C_VEL
LIN {X 0,Y 86.906,Z 465.096,A -85,B 0,C 180,E1 -28183.076,E2 -28183.076} C_VEL
LIN {X 0,Y 86.282,Z 473.507,A -85,B 0,C 180,E1 -28194.034,E2 -28194.034} C_VEL
LIN {X 0,Y 90.217,Z 481.082,A -85,B 0,C 180,E1 -28205.751,E2 -28205.751} C_VEL
LIN {X 0,Y 98.284,Z 487.12,A -85,B 0,C 180,E1 -28215.65,E2 -28215.65} C_VEL
LIN {X 0,Y 99.917,Z 487.618,A -85,B 0,C 180,E1 -28218.071,E2 -28218.071} C_VEL
LIN {X 0,Y 92.186,Z 478.631,A -85,B 0,C 180,E1 -28223.784,E2 -28223.784} C_VEL
LIN {X 0,Y 86.762,Z 469.488,A -85,B 0,C 180,E1 -28229.585,E2 -28229.585} C_VEL
LIN {X 0,Y 82.905,Z 458.871,A -85,B 0,C 180,E1 -28236.255,E2 -28236.255} C_VEL
LIN {X 0,Y 81.008,Z 449.074,A -85,B 0,C 180,E1 -28241.866,E2 -28241.866} C_VEL
LIN {X 0,Y 79.946,Z 436.471,A -85,B 0,C 180,E1 -28247.949,E2 -28247.949} C_VEL
LIN {X 0,Y 79.173,Z 425.431,A -85,B 0,C 180,E1 -28251.899,E2 -28251.899} C_VEL
LIN {X 0,Y 78.827,Z 424.291,A -85,B 0,C 180,E1 -28252.26,E2 -28252.26} C_VEL
LIN {X 0,Y 73.588,Z 420.026,A -85,B 0,C 180,E1 -28260,E2 -28260} C_VEL
LIN {X 0,Y 70.737,Z 414.732,A -85,B 0,C 180,E1 -28271.462,E2 -28271.462} C_VEL
LIN {X 0,Y 70.734,Z 411.677,A -85,B 0,C 180,E1 -28278.84,E2 -28278.84} C_VEL
LIN {X 0,Y 71.802,Z 411.541,A -85,B 0,C 180,E1 -28288.245,E2 -28288.245} C_VEL
LIN {X 0,Y 72.285,Z 411.473,A -85,B 0,C 180,E1 -28295.688,E2 -28295.688} C_VEL
LIN {X 0,Y 72.358,Z 411.472,A -85,B 0,C 180,E1 -28299.01,E2 -28299.01} C_VEL
LIN {X 0,Y 72.263,Z 411.484,A -85,B 0,C 180,E1 -28307.094,E2 -28307.094} C_VEL
LIN {X 0,Y 72.298,Z 411.478,A -85,B 0,C 180,E1 -28314.32,E2 -28314.32} C_VEL
LIN {X 0,Y 72.376,Z 411.462,A -85,B 0,C 180,E1 -28320.953,E2 -28320.953} C_VEL
LIN {X 0,Y 72.396,Z 411.461,A -85,B 0,C 180,E1 -28327.15,E2 -28327.15} C_VEL
LIN {X 0,Y 72.723,Z 411.423,A -85,B 0,C 180,E1 -28335.109,E2 -28335.109} C_VEL
LIN {X 0,Y 72.86,Z 411.404,A -85,B 0,C 180,E1 -28338.876,E2 -28338.876} C_VEL
LIN {X 0,Y 73.574,Z 411.321,A -85,B 0,C 180,E1 -28350,E2 -28350} C_VEL
LIN {X 0,Y 72.894,Z 411.4,A -85,B 0,C 180,E1 -28361.117,E2 -28361.117} C_VEL
LIN {X 0,Y 72.613,Z 411.44,A -85,B 0,C 180,E1 -28366.879,E2 -28366.879} C_VEL
LIN {X 0,Y 72.496,Z 411.445,A -85,B 0,C 180,E1 -28368.237,E2 -28368.237} C_VEL
LIN {X 0,Y 71.59,Z 411.564,A -85,B 0,C 180,E1 -28372.873,E2 -28372.873} C_VEL
LIN {X 0,Y 69.918,Z 411.773,A -85,B 0,C 180,E1 -28377.494,E2 -28377.494} C_VEL
LIN {X 0,Y 65.03,Z 412.362,A -85,B 0,C 180,E1 -28394.29,E2 -28394.29} C_VEL
LIN {X 0,Y 65.201,Z 412.361,A -85,B 0,C 180,E1 -28399.703,E2 -28399.703} C_VEL
LIN {X 0,Y 65.254,Z 412.357,A -85,B 0,C 180,E1 -28409.498,E2 -28409.498} C_VEL
LIN {X 0,Y 65.241,Z 412.349,A -85,B 0,C 180,E1 -28414.475,E2 -28414.475} C_VEL
LIN {X 0,Y 65.652,Z 412.301,A -85,B 0,C 180,E1 -28424.458,E2 -28424.458} C_VEL
LIN {X 0,Y 65.784,Z 412.291,A -85,B 0,C 180,E1 -28427.662,E2 -28427.662} C_VEL
LIN {X 0,Y 66.506,Z 412.192,A -85,B 0,C 180,E1 -28439.999,E2 -28439.999} C_VEL
LIN {X 0,Y 65.784,Z 412.291,A -85,B 0,C 180,E1 -28452.337,E2 -28452.337} C_VEL
LIN {X 0,Y 65.391,Z 412.334,A -85,B 0,C 180,E1 -28458.81,E2 -28458.81} C_VEL
LIN {X 0,Y 65.249,Z 412.348,A -85,B 0,C 180,E1 -28465.521,E2 -28465.521} C_VEL
LIN {X 0,Y 65.218,Z 412.356,A -85,B 0,C 180,E1 -28472.602,E2 -28472.602} C_VEL
LIN {X 0,Y 65.411,Z 412.331,A -85,B 0,C 180,E1 -28481.228,E2 -28481.228} C_VEL
LIN {X 0,Y 66.418,Z 412.21,A -85,B 0,C 180,E1 -28490.589,E2 -28490.589} C_VEL
LIN {X 0,Y 67.349,Z 412.298,A -85,B 0,C 180,E1 -28496.286,E2 -28496.286} C_VEL
LIN {X 0,Y 67.355,Z 413.336,A -85,B 0,C 180,E1 -28498.553,E2 -28498.553} C_VEL
LIN {X 0,Y 67.221,Z 422.702,A -85,B 0,C 180,E1 -28520.978,E2 -28520.978} C_VEL
LIN {X 0,Y 71.411,Z 427.021,A -85,B 0,C 180,E1 -28530,E2 -28530} C_VEL
LIN {X 0,Y 74.626,Z 429.223,A -85,B 0,C 180,E1 -28533.713,E2 -28533.713} C_VEL
LIN {X 0,Y 77.159,Z 441.906,A -85,B 0,C 180,E1 -28537.076,E2 -28537.076} C_VEL
LIN {X 0,Y 79.995,Z 451.785,A -85,B 0,C 180,E1 -28540.12,E2 -28540.12} C_VEL
LIN {X 0,Y 81.601,Z 459.208,A -85,B 0,C 180,E1 -28543.977,E2 -28543.977} C_VEL
LIN {X 0,Y 81.908,Z 460.691,A -85,B 0,C 180,E1 -28544.917,E2 -28544.917} C_VEL
LIN {X 0,Y 81.385,Z 467.427,A -85,B 0,C 180,E1 -28553.753,E2 -28553.753} C_VEL
LIN {X 0,Y 84.539,Z 475.143,A -85,B 0,C 180,E1 -28565.587,E2 -28565.587} C_VEL
LIN {X 0,Y 90.44,Z 480.588,A -85,B 0,C 180,E1 -28574.378,E2 -28574.378} C_VEL
LIN {X 0,Y 92.627,Z 481.94,A -85,B 0,C 180,E1 -28576.932,E2 -28576.932} C_VEL
LIN {X 0,Y 85.068,Z 471.834,A -85,B 0,C 180,E1 -28583.204,E2 -28583.204} C_VEL
LIN {X 0,Y 80.691,Z 463.466,A -85,B 0,C 180,E1 -28588.494,E2 -28588.494} C_VEL
LIN {X 0,Y 76.781,Z 450.841,A -85,B 0,C 180,E1 -28596.254,E2 -28596.254} C_VEL
LIN {X 0,Y 75.194,Z 441.057,A -85,B 0,C 180,E1 -28601.613,E2 -28601.613} C_VEL
LIN {X 0,Y 74.46,Z 432.25,A -85,B 0,C 180,E1 -28605.655,E2 -28605.655} C_VEL
LIN {X 0,Y 73.784,Z 424.7,A -85,B 0,C 180,E1 -28608.497,E2 -28608.497} C_VEL
LIN {X 0,Y 69.044,Z 421.537,A -85,B 0,C 180,E1 -28614.158,E2 -28614.158} C_VEL
LIN {X 0,Y 65.071,Z 417.45,A -85,B 0,C 180,E1 -28623.096,E2 -28623.096} C_VEL
LIN {X 0,Y 63.552,Z 412.571,A -85,B 0,C 180,E1 -28635.228,E2 -28635.228} C_VEL
LIN {X 0,Y 64.367,Z 412.461,A -85,B 0,C 180,E1 -28645.897,E2 -28645.897} C_VEL
LIN {X 0,Y 64.824,Z 412.412,A -85,B 0,C 180,E1 -28649.849,E2 -28649.849} C_VEL
LIN {X 0,Y 64.952,Z 412.383,A -85,B 0,C 180,E1 -28652.753,E2 -28652.753} C_VEL
LIN {X 0,Y 65.232,Z 412.354,A -85,B 0,C 180,E1 -28661.047,E2 -28661.047} C_VEL
LIN {X 0,Y 65.212,Z 412.356,A -85,B 0,C 180,E1 -28669.711,E2 -28669.711} C_VEL
LIN {X 0,Y 65.256,Z 412.348,A -85,B 0,C 180,E1 -28679.498,E2 -28679.498} C_VEL
LIN {X 0,Y 65.241,Z 412.359,A -85,B 0,C 180,E1 -28684.475,E2 -28684.475} C_VEL
LIN {X 0,Y 65.627,Z 412.308,A -85,B 0,C 180,E1 -28694.542,E2 -28694.542} C_VEL
LIN {X 0,Y 65.757,Z 412.285,A -85,B 0,C 180,E1 -28697.657,E2 -28697.657} C_VEL
LIN {X 0,Y 66.497,Z 412.203,A -85,B 0,C 180,E1 -28710,E2 -28710} C_VEL
LIN {X 0,Y 65.798,Z 412.28,A -85,B 0,C 180,E1 -28722.334,E2 -28722.334} C_VEL
LIN {X 0,Y 65.409,Z 412.335,A -85,B 0,C 180,E1 -28728.804,E2 -28728.804} C_VEL
LIN {X 0,Y 65.246,Z 412.358,A -85,B 0,C 180,E1 -28735.522,E2 -28735.522} C_VEL
LIN {X 0,Y 65.199,Z 412.362,A -85,B 0,C 180,E1 -28742.613,E2 -28742.613} C_VEL
LIN {X 0,Y 65.186,Z 412.362,A -85,B 0,C 180,E1 -28750.999,E2 -28750.999} C_VEL
LIN {X 0,Y 65.03,Z 412.362,A -85,B 0,C 180,E1 -28754.29,E2 -28754.29} C_VEL
LIN {X 0,Y 64.65,Z 412.423,A -85,B 0,C 180,E1 -28757.739,E2 -28757.739} C_VEL
LIN {X 0,Y 63.215,Z 412.613,A -85,B 0,C 180,E1 -28762.886,E2 -28762.886} C_VEL
LIN {X 0,Y 60.052,Z 413.002,A -85,B 0,C 180,E1 -28771.793,E2 -28771.793} C_VEL
LIN {X 0,Y 58.392,Z 413.204,A -85,B 0,C 180,E1 -28781.588,E2 -28781.588} C_VEL
LIN {X 0,Y 58.511,Z 413.187,A -85,B 0,C 180,E1 -28783.591,E2 -28783.591} C_VEL
LIN {X 0,Y 58.66,Z 413.177,A -85,B 0,C 180,E1 -28786.135,E2 -28786.135} C_VEL
LIN {X 0,Y 58.826,Z 413.151,A -85,B 0,C 180,E1 -28793.138,E2 -28793.138} C_VEL
LIN {X 0,Y 59.398,Z 413.077,A -85,B 0,C 180,E1 -28799.999,E2 -28799.999} C_VEL
LIN {X 0,Y 58.826,Z 413.151,A -85,B 0,C 180,E1 -28806.861,E2 -28806.861} C_VEL
LIN {X 0,Y 58.538,Z 413.185,A -85,B 0,C 180,E1 -28816.165,E2 -28816.165} C_VEL
LIN {X 0,Y 58.158,Z 413.24,A -85,B 0,C 180,E1 -28828.905,E2 -28828.905} C_VEL
LIN {X 0,Y 58.144,Z 413.241,A -85,B 0,C 180,E1 -28837.183,E2 -28837.183} C_VEL
LIN {X 0,Y 58.667,Z 413.176,A -85,B 0,C 180,E1 -28845.952,E2 -28845.952} C_VEL
LIN {X 0,Y 59.973,Z 413.015,A -85,B 0,C 180,E1 -28855.115,E2 -28855.115} C_VEL
LIN {X 0,Y 60.023,Z 413.087,A -85,B 0,C 180,E1 -28859.535,E2 -28859.535} C_VEL
LIN {X 0,Y 59.78,Z 420.526,A -85,B 0,C 180,E1 -28879.843,E2 -28879.843} C_VEL
LIN {X 0,Y 63.457,Z 424.654,A -85,B 0,C 180,E1 -28890.001,E2 -28890.001} C_VEL
LIN {X 0,Y 67.818,Z 427.677,A -85,B 0,C 180,E1 -28895.949,E2 -28895.949} C_VEL
LIN {X 0,Y 69.848,Z 428.872,A -85,B 0,C 180,E1 -28897.905,E2 -28897.905} C_VEL
LIN {X 0,Y 73.308,Z 443.37,A -85,B 0,C 180,E1 -28901.907,E2 -28901.907} C_VEL
LIN {X 0,Y 75.522,Z 450.196,A -85,B 0,C 180,E1 -28904.049,E2 -28904.049} C_VEL
LIN {X 0,Y 77.094,Z 456.805,A -85,B 0,C 180,E1 -28907.683,E2 -28907.683} C_VEL
LIN {X 0,Y 77.416,Z 464.705,A -85,B 0,C 180,E1 -28918.845,E2 -28918.845} C_VEL
LIN {X 0,Y 81.538,Z 471.734,A -85,B 0,C 180,E1 -28929.952,E2 -28929.952} C_VEL
LIN {X 0,Y 85.007,Z 474.955,A -85,B 0,C 180,E1 -28935.054,E2 -28935.054} C_VEL
LIN {X 0,Y 84.676,Z 474.217,A -85,B 0,C 180,E1 -28936.514,E2 -28936.514} C_VEL
LIN {X 0,Y 77.343,Z 462.323,A -85,B 0,C 180,E1 -28943.798,E2 -28943.798} C_VEL
LIN {X 0,Y 73.213,Z 451.689,A -85,B 0,C 180,E1 -28950.451,E2 -28950.451} C_VEL
LIN {X 0,Y 70.638,Z 439.706,A -85,B 0,C 180,E1 -28957.324,E2 -28957.324} C_VEL
LIN {X 0,Y 69.602,Z 431.087,A -85,B 0,C 180,E1 -28961.607,E2 -28961.607} C_VEL
LIN {X 0,Y 68.897,Z 425.069,A -85,B 0,C 180,E1 -28964.014,E2 -28964.014} C_VEL
LIN {X 0,Y 61.512,Z 420.231,A -85,B 0,C 180,E1 -28973.44,E2 -28973.44} C_VEL
LIN {X 0,Y 56.829,Z 414.424,A -85,B 0,C 180,E1 -28988.364,E2 -28988.364} C_VEL
LIN {X 0,Y 56.543,Z 413.441,A -85,B 0,C 180,E1 -28991.735,E2 -28991.735} C_VEL
LIN {X 0,Y 56.815,Z 413.409,A -85,B 0,C 180,E1 -29001.784,E2 -29001.784} C_VEL
LIN {X 0,Y 57.633,Z 413.307,A -85,B 0,C 180,E1 -29009.195,E2 -29009.195} C_VEL
LIN {X 0,Y 57.845,Z 413.274,A -85,B 0,C 180,E1 -29011.735,E2 -29011.735} C_VEL
LIN {X 0,Y 57.962,Z 413.263,A -85,B 0,C 180,E1 -29017.32,E2 -29017.32} C_VEL
LIN {X 0,Y 58.07,Z 413.243,A -85,B 0,C 180,E1 -29023.433,E2 -29023.433} C_VEL
LIN {X 0,Y 58.037,Z 413.248,A -85,B 0,C 180,E1 -29032.736,E2 -29032.736} C_VEL
LIN {X 0,Y 58.16,Z 413.236,A -85,B 0,C 180,E1 -29037.768,E2 -29037.768} C_VEL
LIN {X 0,Y 58.152,Z 413.233,A -85,B 0,C 180,E1 -29041.09,E2 -29041.09} C_VEL
LIN {X 0,Y 58.518,Z 413.195,A -85,B 0,C 180,E1 -29053.906,E2 -29053.906} C_VEL
LIN {X 0,Y 58.802,Z 413.158,A -85,B 0,C 180,E1 -29063.135,E2 -29063.135} C_VEL
LIN {X 0,Y 59.387,Z 413.088,A -85,B 0,C 180,E1 -29069.999,E2 -29069.999} C_VEL
LIN {X 0,Y 58.826,Z 413.154,A -85,B 0,C 180,E1 -29076.861,E2 -29076.861} C_VEL
LIN {X 0,Y 58.677,Z 413.167,A -85,B 0,C 180,E1 -29083.859,E2 -29083.859} C_VEL
LIN {X 0,Y 58.205,Z 413.225,A -85,B 0,C 180,E1 -29091.237,E2 -29091.237} C_VEL
LIN {X 0,Y 58.154,Z 413.233,A -85,B 0,C 180,E1 -29098.908,E2 -29098.908} C_VEL
LIN {X 0,Y 58.16,Z 413.236,A -85,B 0,C 180,E1 -29102.233,E2 -29102.233} C_VEL
LIN {X 0,Y 58.034,Z 413.248,A -85,B 0,C 180,E1 -29107.265,E2 -29107.265} C_VEL
LIN {X 0,Y 58.012,Z 413.25,A -85,B 0,C 180,E1 -29116.625,E2 -29116.625} C_VEL
LIN {X 0,Y 58.031,Z 413.255,A -85,B 0,C 180,E1 -29122.731,E2 -29122.731} C_VEL
LIN {X 0,Y 58.158,Z 413.236,A -85,B 0,C 180,E1 -29127.769,E2 -29127.769} C_VEL
LIN {X 0,Y 58.152,Z 413.24,A -85,B 0,C 180,E1 -29131.09,E2 -29131.09} C_VEL
LIN {X 0,Y 58.511,Z 413.187,A -85,B 0,C 180,E1 -29143.591,E2 -29143.591} C_VEL
LIN {X 0,Y 58.311,Z 413.222,A -85,B 0,C 180,E1 -29146.742,E2 -29146.742} C_VEL
LIN {X 0,Y 56.823,Z 413.406,A -85,B 0,C 180,E1 -29151.065,E2 -29151.065} C_VEL
LIN {X 0,Y 51.983,Z 414.009,A -85,B 0,C 180,E1 -29163.2,E2 -29163.2} C_VEL
LIN {X 0,Y 51.814,Z 414.007,A -85,B 0,C 180,E1 -29164.732,E2 -29164.732} C_VEL
LIN {X 0,Y 51.483,Z 414.064,A -85,B 0,C 180,E1 -29175.844,E2 -29175.844} C_VEL
LIN {X 0,Y 51.03,Z 414.12,A -85,B 0,C 180,E1 -29184.403,E2 -29184.403} C_VEL
LIN {X 0,Y 51.077,Z 414.113,A -85,B 0,C 180,E1 -29194.353,E2 -29194.353} C_VEL
LIN {X 0,Y 51.716,Z 414.044,A -85,B 0,C 180,E1 -29207.198,E2 -29207.198} C_VEL
LIN {X 0,Y 52.515,Z 413.942,A -85,B 0,C 180,E1 -29213.414,E2 -29213.414} C_VEL
LIN {X 0,Y 53.059,Z 413.873,A -85,B 0,C 180,E1 -29218.007,E2 -29218.007} C_VEL
LIN {X 0,Y 52.149,Z 414.162,A -85,B 0,C 180,E1 -29225.093,E2 -29225.093} C_VEL
LIN {X 0,Y 54.274,Z 421,A -85,B 0,C 180,E1 -29246.288,E2 -29246.288} C_VEL
LIN {X 0,Y 59.656,Z 425.2,A -85,B 0,C 180,E1 -29256.766,E2 -29256.766} C_VEL
LIN {X 0,Y 65.625,Z 428.521,A -85,B 0,C 180,E1 -29262.722,E2 -29262.722} C_VEL
LIN {X 0,Y 69.014,Z 441.463,A -85,B 0,C 180,E1 -29266.263,E2 -29266.263} C_VEL
LIN {X 0,Y 71.318,Z 447.99,A -85,B 0,C 180,E1 -29268.18,E2 -29268.18} C_VEL
LIN {X 0,Y 72.649,Z 452.665,A -85,B 0,C 180,E1 -29270.772,E2 -29270.772} C_VEL
LIN {X 0,Y 73.377,Z 459.969,A -85,B 0,C 180,E1 -29281.467,E2 -29281.467} C_VEL
LIN {X 0,Y 77.858,Z 466.956,A -85,B 0,C 180,E1 -29292.614,E2 -29292.614} C_VEL
LIN {X 0,Y 78.922,Z 468.013,A -85,B 0,C 180,E1 -29294.57,E2 -29294.57} C_VEL
LIN {X 0,Y 72.361,Z 456.546,A -85,B 0,C 180,E1 -29301.479,E2 -29301.479} C_VEL
LIN {X 0,Y 68.004,Z 444.595,A -85,B 0,C 180,E1 -29308.887,E2 -29308.887} C_VEL
LIN {X 0,Y 65.674,Z 432.546,A -85,B 0,C 180,E1 -29315.502,E2 -29315.502} C_VEL
LIN {X 0,Y 64.687,Z 425.488,A -85,B 0,C 180,E1 -29318.698,E2 -29318.698} C_VEL
LIN {X 0,Y 54.029,Z 418.883,A -85,B 0,C 180,E1 -29332.527,E2 -29332.527} C_VEL
LIN {X 0,Y 49.989,Z 414.256,A -85,B 0,C 180,E1 -29346.053,E2 -29346.053} C_VEL
LIN {X 0,Y 49.98,Z 414.252,A -85,B 0,C 180,E1 -29364.952,E2 -29364.952} C_VEL
LIN {X 0,Y 50.78,Z 414.148,A -85,B 0,C 180,E1 -29373.858,E2 -29373.858} C_VEL
LIN {X 0,Y 51.033,Z 414.119,A -85,B 0,C 180,E1 -29383.519,E2 -29383.519} C_VEL
LIN {X 0,Y 51.024,Z 414.129,A -85,B 0,C 180,E1 -29386.472,E2 -29386.472} C_VEL
LIN {X 0,Y 51.053,Z 414.125,A -85,B 0,C 180,E1 -29396.588,E2 -29396.588} C_VEL
LIN {X 0,Y 51.025,Z 414.127,A -85,B 0,C 180,E1 -29405.592,E2 -29405.592} C_VEL
LIN {X 0,Y 51.459,Z 414.073,A -85,B 0,C 180,E1 -29414.148,E2 -29414.148} C_VEL
LIN {X 0,Y 51.679,Z 414.047,A -85,B 0,C 180,E1 -29422.183,E2 -29422.183} C_VEL
LIN {X 0,Y 52.27,Z 413.975,A -85,B 0,C 180,E1 -29429.999,E2 -29429.999} C_VEL
LIN {X 0,Y 51.705,Z 414.044,A -85,B 0,C 180,E1 -29437.811,E2 -29437.811} C_VEL
LIN {X 0,Y 51.419,Z 414.08,A -85,B 0,C 180,E1 -29446.906,E2 -29446.906} C_VEL
LIN {X 0,Y 51.032,Z 414.126,A -85,B 0,C 180,E1 -29454.402,E2 -29454.402} C_VEL
LIN {X 0,Y 51.031,Z 414.129,A -85,B 0,C 180,E1 -29464.276,E2 -29464.276} C_VEL
LIN {X 0,Y 50.979,Z 414.126,A -85,B 0,C 180,E1 -29476.424,E2 -29476.424} C_VEL
LIN {X 0,Y 51.049,Z 414.117,A -85,B 0,C 180,E1 -29486.585,E2 -29486.585} C_VEL
LIN {X 0,Y 51.027,Z 414.121,A -85,B 0,C 180,E1 -29495.593,E2 -29495.593} C_VEL
LIN {X 0,Y 51.483,Z 414.064,A -85,B 0,C 180,E1 -29504.155,E2 -29504.155} C_VEL
LIN {X 0,Y 51.702,Z 414.036,A -85,B 0,C 180,E1 -29512.187,E2 -29512.187} C_VEL
LIN {X 0,Y 52.283,Z 413.963,A -85,B 0,C 180,E1 -29519.999,E2 -29519.999} C_VEL
LIN {X 0,Y 51.814,Z 414.007,A -85,B 0,C 180,E1 -29524.732,E2 -29524.732} C_VEL
LIN {X 0,Y 51.24,Z 414.093,A -85,B 0,C 180,E1 -29529.047,E2 -29529.047} C_VEL
LIN {X 0,Y 49.58,Z 414.315,A -85,B 0,C 180,E1 -29535.506,E2 -29535.506} C_VEL
LIN {X 0,Y 47.504,Z 414.585,A -85,B 0,C 180,E1 -29542.124,E2 -29542.124} C_VEL
LIN {X 0,Y 44.242,Z 414.973,A -85,B 0,C 180,E1 -29557.137,E2 -29557.137} C_VEL
LIN {X 0,Y 44.126,Z 414.965,A -85,B 0,C 180,E1 -29562.497,E2 -29562.497} C_VEL
LIN {X 0,Y 45.07,Z 414.863,A -85,B 0,C 180,E1 -29571.411,E2 -29571.411} C_VEL
LIN {X 0,Y 45.327,Z 414.836,A -85,B 0,C 180,E1 -29582.281,E2 -29582.281} C_VEL
LIN {X 0,Y 44.918,Z 414.921,A -85,B 0,C 180,E1 -29591.765,E2 -29591.765} C_VEL
LIN {X 0,Y 49.267,Z 421.087,A -85,B 0,C 180,E1 -29613.078,E2 -29613.078} C_VEL
LIN {X 0,Y 54.2,Z 424.234,A -85,B 0,C 180,E1 -29621.216,E2 -29621.216} C_VEL
LIN {X 0,Y 62.164,Z 428.221,A -85,B 0,C 180,E1 -29628.274,E2 -29628.274} C_VEL
LIN {X 0,Y 66.103,Z 441.545,A -85,B 0,C 180,E1 -29631.847,E2 -29631.847} C_VEL
LIN {X 0,Y 67.653,Z 445.568,A -85,B 0,C 180,E1 -29632.928,E2 -29632.928} C_VEL
LIN {X 0,Y 68.555,Z 448.246,A -85,B 0,C 180,E1 -29634.21,E2 -29634.21} C_VEL
LIN {X 0,Y 69.618,Z 454.641,A -85,B 0,C 180,E1 -29643.727,E2 -29643.727} C_VEL
LIN {X 0,Y 72.829,Z 460.068,A -85,B 0,C 180,E1 -29652.494,E2 -29652.494} C_VEL
LIN {X 0,Y 72.596,Z 459.623,A -85,B 0,C 180,E1 -29653.289,E2 -29653.289} C_VEL
LIN {X 0,Y 67.341,Z 449.324,A -85,B 0,C 180,E1 -29659.5,E2 -29659.5} C_VEL
LIN {X 0,Y 63.505,Z 437.833,A -85,B 0,C 180,E1 -29666.404,E2 -29666.404} C_VEL
LIN {X 0,Y 61.423,Z 427.697,A -85,B 0,C 180,E1 -29671.838,E2 -29671.838} C_VEL
LIN {X 0,Y 61.138,Z 425.879,A -85,B 0,C 180,E1 -29672.625,E2 -29672.625} C_VEL
LIN {X 0,Y 55.818,Z 423.089,A -85,B 0,C 180,E1 -29677.808,E2 -29677.808} C_VEL
LIN {X 0,Y 48.492,Z 418.858,A -85,B 0,C 180,E1 -29687.444,E2 -29687.444} C_VEL
LIN {X 0,Y 43.875,Z 415.015,A -85,B 0,C 180,E1 -29700.001,E2 -29700.001} C_VEL
LIN {X 0,Y 42.47,Z 415.191,A -85,B 0,C 180,E1 -29719.328,E2 -29719.328} C_VEL
LIN {X 0,Y 43.153,Z 415.11,A -85,B 0,C 180,E1 -29729.249,E2 -29729.249} C_VEL
LIN {X 0,Y 43.691,Z 415.035,A -85,B 0,C 180,E1 -29736.456,E2 -29736.456} C_VEL
LIN {X 0,Y 43.748,Z 415.032,A -85,B 0,C 180,E1 -29739.987,E2 -29739.987} C_VEL
LIN {X 0,Y 43.826,Z 415.017,A -85,B 0,C 180,E1 -29750.099,E2 -29750.099} C_VEL
LIN {X 0,Y 43.845,Z 415.015,A -85,B 0,C 180,E1 -29761.256,E2 -29761.256} C_VEL
LIN {X 0,Y 44.23,Z 414.976,A -85,B 0,C 180,E1 -29772.44,E2 -29772.44} C_VEL
LIN {X 0,Y 44.532,Z 414.938,A -85,B 0,C 180,E1 -29780.919,E2 -29780.919} C_VEL
LIN {X 0,Y 45.144,Z 414.862,A -85,B 0,C 180,E1 -29789.999,E2 -29789.999} C_VEL
LIN {X 0,Y 44.562,Z 414.934,A -85,B 0,C 180,E1 -29799.074,E2 -29799.074} C_VEL
LIN {X 0,Y 44.202,Z 414.976,A -85,B 0,C 180,E1 -29808.541,E2 -29808.541} C_VEL
LIN {X 0,Y 43.848,Z 415.014,A -85,B 0,C 180,E1 -29818.74,E2 -29818.74} C_VEL
LIN {X 0,Y 43.802,Z 415.02,A -85,B 0,C 180,E1 -29829.925,E2 -29829.925} C_VEL
LIN {X 0,Y 43.825,Z 415.021,A -85,B 0,C 180,E1 -29843.303,E2 -29843.303} C_VEL
LIN {X 0,Y 43.844,Z 415.021,A -85,B 0,C 180,E1 -29851.255,E2 -29851.255} C_VEL
LIN {X 0,Y 44.258,Z 414.962,A -85,B 0,C 180,E1 -29862.319,E2 -29862.319} C_VEL
LIN {X 0,Y 44.553,Z 414.925,A -85,B 0,C 180,E1 -29870.923,E2 -29870.923} C_VEL
LIN {X 0,Y 45.159,Z 414.85,A -85,B 0,C 180,E1 -29879.999,E2 -29879.999} C_VEL
LIN {X 0,Y 44.553,Z 414.926,A -85,B 0,C 180,E1 -29889.075,E2 -29889.075} C_VEL
LIN {X 0,Y 44.195,Z 414.971,A -85,B 0,C 180,E1 -29898.544,E2 -29898.544} C_VEL
LIN {X 0,Y 43.861,Z 415.019,A -85,B 0,C 180,E1 -29908.731,E2 -29908.731} C_VEL
LIN {X 0,Y 44.051,Z 414.996,A -85,B 0,C 180,E1 -29919.655,E2 -29919.655} C_VEL
LIN {X 0,Y 44.126,Z 414.965,A -85,B 0,C 180,E1 -29922.497,E2 -29922.497} C_VEL
LIN {X 0,Y 43.648,Z 415.048,A -85,B 0,C 180,E1 -29927.501,E2 -29927.501} C_VEL
LIN {X 0,Y 42.265,Z 415.22,A -85,B 0,C 180,E1 -29932.435,E2 -29932.435} C_VEL
LIN {X 0,Y 37.886,Z 415.759,A -85,B 0,C 180,E1 -29949.201,E2 -29949.201} C_VEL
LIN {X 0,Y 37.835,Z 415.748,A -85,B 0,C 180,E1 -29951.313,E2 -29951.313} C_VEL
LIN {X 0,Y 38.664,Z 415.753,A -85,B 0,C 180,E1 -29961.508,E2 -29961.508} C_VEL
LIN {X 0,Y 44.078,Z 420.458,A -85,B 0,C 180,E1 -29979.175,E2 -29979.175} C_VEL
LIN {X 0,Y 52.248,Z 424.724,A -85,B 0,C 180,E1 -29989.681,E2 -29989.681} C_VEL
LIN {X 0,Y 59.367,Z 427.952,A -85,B 0,C 180,E1 -29994.478,E2 -29994.478} C_VEL
LIN {X 0,Y 63.435,Z 440.47,A -85,B 0,C 180,E1 -29997.586,E2 -29997.586} C_VEL
LIN {X 0,Y 64.969,Z 444.319,A -85,B 0,C 180,E1 -29998.676,E2 -29998.676} C_VEL
LIN {X 0,Y 67.004,Z 450.8,A -85,B 0,C 180,E1 -30009.002,E2 -30009.002} C_VEL
LIN {X 0,Y 67.69,Z 451.987,A -85,B 0,C 180,E1 -30011.086,E2 -30011.086} C_VEL
LIN {X 0,Y 62.54,Z 440.922,A -85,B 0,C 180,E1 -30017.604,E2 -30017.604} C_VEL
LIN {X 0,Y 58.964,Z 428.643,A -85,B 0,C 180,E1 -30024.476,E2 -30024.476} C_VEL
LIN {X 0,Y 58.475,Z 426.283,A -85,B 0,C 180,E1 -30025.711,E2 -30025.711} C_VEL
LIN {X 0,Y 51.688,Z 423.01,A -85,B 0,C 180,E1 -30031.62,E2 -30031.62} C_VEL
LIN {X 0,Y 43.425,Z 418.779,A -85,B 0,C 180,E1 -30041.115,E2 -30041.115} C_VEL
LIN {X 0,Y 38.672,Z 415.65,A -85,B 0,C 180,E1 -30051.51,E2 -30051.51} C_VEL
LIN {X 0,Y 35.533,Z 416.053,A -85,B 0,C 180,E1 -30083.303,E2 -30083.303} C_VEL
LIN {X 0,Y 36.451,Z 415.935,A -85,B 0,C 180,E1 -30095.341,E2 -30095.341} C_VEL
LIN {X 0,Y 36.704,Z 415.908,A -85,B 0,C 180,E1 -30100.011,E2 -30100.011} C_VEL
LIN {X 0,Y 36.737,Z 415.9,A -85,B 0,C 180,E1 -30109.928,E2 -30109.928} C_VEL
LIN {X 0,Y 36.73,Z 415.908,A -85,B 0,C 180,E1 -30114.968,E2 -30114.968} C_VEL
LIN {X 0,Y 37.056,Z 415.865,A -85,B 0,C 180,E1 -30131.496,E2 -30131.496} C_VEL
LIN {X 0,Y 37.329,Z 415.828,A -85,B 0,C 180,E1 -30139.147,E2 -30139.147} C_VEL
LIN {X 0,Y 38.002,Z 415.752,A -85,B 0,C 180,E1 -30149.999,E2 -30149.999} C_VEL
LIN {X 0,Y 37.358,Z 415.824,A -85,B 0,C 180,E1 -30160.843,E2 -30160.843} C_VEL
LIN {X 0,Y 37.085,Z 415.861,A -85,B 0,C 180,E1 -30168.637,E2 -30168.637} C_VEL
LIN {X 0,Y 36.725,Z 415.909,A -85,B 0,C 180,E1 -30185.036,E2 -30185.036} C_VEL
LIN {X 0,Y 36.723,Z 415.902,A -85,B 0,C 180,E1 -30190.045,E2 -30190.045} C_VEL
LIN {X 0,Y 36.716,Z 415.907,A -85,B 0,C 180,E1 -30199.965,E2 -30199.965} C_VEL
LIN {X 0,Y 36.711,Z 415.902,A -85,B 0,C 180,E1 -30204.946,E2 -30204.946} C_VEL
LIN {X 0,Y 37.08,Z 415.857,A -85,B 0,C 180,E1 -30221.381,E2 -30221.381} C_VEL
LIN {X 0,Y 37.351,Z 415.826,A -85,B 0,C 180,E1 -30229.153,E2 -30229.153} C_VEL
LIN {X 0,Y 38.018,Z 415.739,A -85,B 0,C 180,E1 -30239.999,E2 -30239.999} C_VEL
LIN {X 0,Y 37.351,Z 415.826,A -85,B 0,C 180,E1 -30250.845,E2 -30250.845} C_VEL
LIN {X 0,Y 37.082,Z 415.857,A -85,B 0,C 180,E1 -30258.627,E2 -30258.627} C_VEL
LIN {X 0,Y 36.819,Z 415.889,A -85,B 0,C 180,E1 -30274.934,E2 -30274.934} C_VEL
LIN {X 0,Y 37.534,Z 415.806,A -85,B 0,C 180,E1 -30288.5,E2 -30288.5} C_VEL
LIN {X 0,Y 37.949,Z 415.758,A -85,B 0,C 180,E1 -30296.25,E2 -30296.25} C_VEL
LIN {X 0,Y 37.846,Z 415.764,A -85,B 0,C 180,E1 -30308.199,E2 -30308.199} C_VEL
LIN {X 0,Y 37.835,Z 415.748,A -85,B 0,C 180,E1 -30311.313,E2 -30311.313} C_VEL
LIN {X 0,Y 37.486,Z 415.831,A -85,B 0,C 180,E1 -30317.411,E2 -30317.411} C_VEL
LIN {X 0,Y 36.189,Z 416.433,A -85,B 0,C 180,E1 -30327.771,E2 -30327.771} C_VEL
LIN {X 0,Y 36.209,Z 417.719,A -85,B 0,C 180,E1 -30338.267,E2 -30338.267} C_VEL
LIN {X 0,Y 37.775,Z 418.86,A -85,B 0,C 180,E1 -30343.652,E2 -30343.652} C_VEL
LIN {X 0,Y 46.464,Z 423.004,A -85,B 0,C 180,E1 -30354.833,E2 -30354.833} C_VEL
LIN {X 0,Y 55.492,Z 426.741,A -85,B 0,C 180,E1 -30360.438,E2 -30360.438} C_VEL
LIN {X 0,Y 57.365,Z 427.492,A -85,B 0,C 180,E1 -30361.175,E2 -30361.175} C_VEL
LIN {X 0,Y 61.932,Z 440.013,A -85,B 0,C 180,E1 -30363.923,E2 -30363.923} C_VEL
LIN {X 0,Y 62.173,Z 440.682,A -85,B 0,C 180,E1 -30364.417,E2 -30364.417} C_VEL
LIN {X 0,Y 63.133,Z 443.398,A -85,B 0,C 180,E1 -30368.809,E2 -30368.809} C_VEL
LIN {X 0,Y 58.445,Z 432.318,A -85,B 0,C 180,E1 -30375.052,E2 -30375.052} C_VEL
LIN {X 0,Y 56.614,Z 426.592,A -85,B 0,C 180,E1 -30378.146,E2 -30378.146} C_VEL
LIN {X 0,Y 51.42,Z 424.278,A -85,B 0,C 180,E1 -30382.045,E2 -30382.045} C_VEL
LIN {X 0,Y 35.21,Z 416.61,A -85,B 0,C 180,E1 -30399.556,E2 -30399.556} C_VEL
LIN {X 0,Y 34.084,Z 416.229,A -85,B 0,C 180,E1 -30401.984,E2 -30401.984} C_VEL
LIN {X 0,Y 28.241,Z 416.79,A -85,B 0,C 180,E1 -30434.411,E2 -30434.411} C_VEL
LIN {X 0,Y 28.696,Z 416.749,A -85,B 0,C 180,E1 -30449.331,E2 -30449.331} C_VEL
LIN {X 0,Y 29.541,Z 416.668,A -85,B 0,C 180,E1 -30465.541,E2 -30465.541} C_VEL
LIN {X 0,Y 29.499,Z 416.672,A -85,B 0,C 180,E1 -30481.542,E2 -30481.542} C_VEL
LIN {X 0,Y 29.865,Z 416.638,A -85,B 0,C 180,E1 -30490.277,E2 -30490.277} C_VEL
LIN {X 0,Y 30.106,Z 416.614,A -85,B 0,C 180,E1 -30496.499,E2 -30496.499} C_VEL
LIN {X 0,Y 30.819,Z 416.551,A -85,B 0,C 180,E1 -30509.999,E2 -30509.999} C_VEL
LIN {X 0,Y 30.134,Z 416.611,A -85,B 0,C 180,E1 -30523.486,E2 -30523.486} C_VEL
LIN {X 0,Y 29.894,Z 416.634,A -85,B 0,C 180,E1 -30529.878,E2 -30529.878} C_VEL
LIN {X 0,Y 29.512,Z 416.67,A -85,B 0,C 180,E1 -30538.442,E2 -30538.442} C_VEL
LIN {X 0,Y 29.538,Z 416.668,A -85,B 0,C 180,E1 -30555.543,E2 -30555.543} C_VEL
LIN {X 0,Y 29.503,Z 416.673,A -85,B 0,C 180,E1 -30571.546,E2 -30571.546} C_VEL
LIN {X 0,Y 29.889,Z 416.636,A -85,B 0,C 180,E1 -30580.139,E2 -30580.139} C_VEL
LIN {X 0,Y 30.128,Z 416.615,A -85,B 0,C 180,E1 -30586.509,E2 -30586.509} C_VEL
LIN {X 0,Y 30.837,Z 416.545,A -85,B 0,C 180,E1 -30599.999,E2 -30599.999} C_VEL
LIN {X 0,Y 30.128,Z 416.615,A -85,B 0,C 180,E1 -30613.488,E2 -30613.488} C_VEL
LIN {X 0,Y 29.893,Z 416.636,A -85,B 0,C 180,E1 -30619.88,E2 -30619.88} C_VEL
LIN {X 0,Y 29.584,Z 416.665,A -85,B 0,C 180,E1 -30628.366,E2 -30628.366} C_VEL
LIN {X 0,Y 30.156,Z 416.612,A -85,B 0,C 180,E1 -30645.642,E2 -30645.642} C_VEL
LIN {X 0,Y 30.66,Z 416.564,A -85,B 0,C 180,E1 -30662.714,E2 -30662.714} C_VEL
LIN {X 0,Y 33.901,Z 416.371,A -85,B 0,C 180,E1 -30693.589,E2 -30693.589} C_VEL
LIN {X 0,Y 37.775,Z 418.86,A -85,B 0,C 180,E1 -30703.652,E2 -30703.652} C_VEL
LIN {X 0,Y 39.769,Z 420.038,A -85,B 0,C 180,E1 -30708.559,E2 -30708.559} C_VEL
LIN {X 0,Y 46.316,Z 423.279,A -85,B 0,C 180,E1 -30723.773,E2 -30723.773} C_VEL
LIN {X 0,Y 49.491,Z 424.506,A -85,B 0,C 180,E1 -30726.113,E2 -30726.113} C_VEL
LIN {X 0,Y 56.468,Z 427.16,A -85,B 0,C 180,E1 -30728.298,E2 -30728.298} C_VEL
LIN {X 0,Y 56.617,Z 427.553,A -85,B 0,C 180,E1 -30728.366,E2 -30728.366} C_VEL
LIN {X 0,Y 56.569,Z 427.554,A -85,B 0,C 180,E1 -30729.672,E2 -30729.672} C_VEL
LIN {X 0,Y 56.008,Z 426.923,A -85,B 0,C 180,E1 -30730.08,E2 -30730.08} C_VEL
LIN {X 0,Y 49.049,Z 424.073,A -85,B 0,C 180,E1 -30734.241,E2 -30734.241} C_VEL
LIN {X 0,Y 30.916,Z 416.541,A -85,B 0,C 180,E1 -30749.594,E2 -30749.594} C_VEL
LIN {X 0,Y 24.921,Z 417,A -85,B 0,C 180,E1 -30763.621,E2 -30763.621} C_VEL
LIN {X 0,Y 21.101,Z 417.118,A -85,B 0,C 180,E1 -30799.457,E2 -30799.457} C_VEL
LIN {X 0,Y 21.886,Z 417.094,A -85,B 0,C 180,E1 -30819.961,E2 -30819.961} C_VEL
LIN {X 0,Y 22.195,Z 417.085,A -85,B 0,C 180,E1 -30830.705,E2 -30830.705} C_VEL
LIN {X 0,Y 22.813,Z 417.065,A -85,B 0,C 180,E1 -30852.055,E2 -30852.055} C_VEL
LIN {X 0,Y 23.588,Z 417.041,A -85,B 0,C 180,E1 -30869.999,E2 -30869.999} C_VEL
LIN {X 0,Y 22.846,Z 417.064,A -85,B 0,C 180,E1 -30887.915,E2 -30887.915} C_VEL
LIN {X 0,Y 22.198,Z 417.084,A -85,B 0,C 180,E1 -30909.287,E2 -30909.287} C_VEL
LIN {X 0,Y 22.195,Z 417.085,A -85,B 0,C 180,E1 -30920.703,E2 -30920.703} C_VEL
LIN {X 0,Y 22.841,Z 417.064,A -85,B 0,C 180,E1 -30942.078,E2 -30942.078} C_VEL
LIN {X 0,Y 23.605,Z 417.041,A -85,B 0,C 180,E1 -30959.999,E2 -30959.999} C_VEL
LIN {X 0,Y 22.845,Z 417.064,A -85,B 0,C 180,E1 -30977.916,E2 -30977.916} C_VEL
LIN {X 0,Y 22.529,Z 417.074,A -85,B 0,C 180,E1 -30998.6,E2 -30998.6} C_VEL
LIN {X 0,Y 22.948,Z 417.061,A -85,B 0,C 180,E1 -31012.23,E2 -31012.23} C_VEL
LIN {X 0,Y 23.518,Z 417.043,A -85,B 0,C 180,E1 -31023.7,E2 -31023.7} C_VEL
LIN {X 0,Y 30.665,Z 416.674,A -85,B 0,C 180,E1 -31067.507,E2 -31067.507} C_VEL
LIN {X 0,Y 41.14,Z 421.257,A -85,B 0,C 180,E1 -31081.335,E2 -31081.335} C_VEL
LIN {X 0,Y 49.491,Z 424.506,A -85,B 0,C 180,E1 -31086.113,E2 -31086.113} C_VEL
LIN {X 0,Y 47.445,Z 423.941,A -85,B 0,C 180,E1 -31086.639,E2 -31086.639} C_VEL
LIN {X 0,Y 41.631,Z 422.071,A -85,B 0,C 180,E1 -31085.956,E2 -31085.956} C_VEL
LIN {X 0,Y 30.857,Z 418.719,A -85,B 0,C 180,E1 -31081.719,E2 -31081.719} C_VEL
LIN {X 0,Y 24.618,Z 417.348,A -85,B 0,C 180,E1 -31075.23,E2 -31075.23} C_VEL
LIN {X 0,Y 21.473,Z 417.103,A -85,B 0,C 180,E1 -31068.124,E2 -31068.124} C_VEL
LIN {X 0,Y 16.307,Z 417.178,A -85,B 0,C 180,E1 -31024.472,E2 -31024.472} C_VEL
LIN {X 0,Y 15.369,Z 417.178,A -85,B 0,C 180,E1 -30983.861,E2 -30983.861} C_VEL
LIN {X 0,Y 16.277,Z 417.178,A -85,B 0,C 180,E1 -30959.998,E2 -30959.998} C_VEL
LIN {X 0,Y 15.286,Z 417.178,A -85,B 0,C 180,E1 -30936.849,E2 -30936.849} C_VEL
LIN {X 0,Y 15.107,Z 417.178,A -85,B 0,C 180,E1 -30932.272,E2 -30932.272} C_VEL
LIN {X 0,Y 15.111,Z 417.178,A -85,B 0,C 180,E1 -30897.714,E2 -30897.714} C_VEL
LIN {X 0,Y 15.29,Z 417.178,A -85,B 0,C 180,E1 -30893.17,E2 -30893.17} C_VEL
LIN {X 0,Y 16.257,Z 417.178,A -85,B 0,C 180,E1 -30869.998,E2 -30869.998} C_VEL
LIN {X 0,Y 15.258,Z 417.178,A -85,B 0,C 180,E1 -30847.107,E2 -30847.107} C_VEL
LIN {X 0,Y 14.796,Z 417.178,A -85,B 0,C 180,E1 -30823.471,E2 -30823.471} C_VEL
LIN {X 0,Y 14.179,Z 417.178,A -85,B 0,C 180,E1 -30787.53,E2 -30787.53} C_VEL
LIN {X 0,Y 26.824,Z 416.918,A -85,B 0,C 180,E1 -30738.079,E2 -30738.079} C_VEL
LIN {X 0,Y 29.846,Z 416.848,A -85,B 0,C 180,E1 -30735.056,E2 -30735.056} C_VEL
LIN {X 0,Y 36.882,Z 419.62,A -85,B 0,C 180,E1 -30730.341,E2 -30730.341} C_VEL
LIN {X 0,Y 36.389,Z 419.453,A -85,B 0,C 180,E1 -30729.418,E2 -30729.418} C_VEL
LIN {X 0,Y 28.735,Z 416.744,A -85,B 0,C 180,E1 -30722.346,E2 -30722.346} C_VEL
LIN {X 0,Y 21.473,Z 417.103,A -85,B 0,C 180,E1 -30708.124,E2 -30708.124} C_VEL
LIN {X 0,Y 18.644,Z 417.178,A -85,B 0,C 180,E1 -30700.373,E2 -30700.373} C_VEL
LIN {X 0,Y 15.46,Z 417.181,A -85,B 0,C 180,E1 -30692.381,E2 -30692.381} C_VEL
LIN {X 0,Y 7.983,Z 417.178,A -85,B 0,C 180,E1 -30630.098,E2 -30630.098} C_VEL
LIN {X 0,Y 8.708,Z 417.178,A -85,B 0,C 180,E1 -30599.996,E2 -30599.996} C_VEL
LIN {X 0,Y 7.781,Z 417.178,A -85,B 0,C 180,E1 -30574.577,E2 -30574.577} C_VEL
LIN {X 0,Y 7.783,Z 417.178,A -85,B 0,C 180,E1 -30535.428,E2 -30535.428} C_VEL
LIN {X 0,Y 8.686,Z 417.178,A -85,B 0,C 180,E1 -30509.996,E2 -30509.996} C_VEL
LIN {X 0,Y 7.856,Z 417.178,A -85,B 0,C 180,E1 -30483.475,E2 -30483.475} C_VEL
LIN {X 0,Y 7.186,Z 417.178,A -85,B 0,C 180,E1 -30420.005,E2 -30420.005} C_VEL
LIN {X 0,Y 18.02,Z 417.178,A -85,B 0,C 180,E1 -30368.738,E2 -30368.738} C_VEL
LIN {X 0,Y 16.653,Z 417.178,A -85,B 0,C 180,E1 -30363.959,E2 -30363.959} C_VEL
LIN {X 0,Y 10.004,Z 417.178,A -85,B 0,C 180,E1 -30330.003,E2 -30330.003} C_VEL
LIN {X 0,Y 8.307,Z 417.178,A -85,B 0,C 180,E1 -30297.776,E2 -30297.776} C_VEL
LIN {X 0,Y 7.983,Z 417.178,A -85,B 0,C 180,E1 -30270.098,E2 -30270.098} C_VEL
LIN {X 0,Y 8.535,Z 419.178,A -85,B 0,C 180,E1 -30256.725,E2 -30256.725} C_VEL
LIN {X 0,Y 8.535,Z 600,A -85,B 0,C 180,E1 -30256.725,E2 -30256.725} C_VEL
LIN {X 0,Y 8.535,Z 600,A -85,B 0,C 180,E1 -30256.725,E2 -30256.725}

QRS_NEXT_CUT()

QRS_NEXT()
QRS_HOME()

END
